LIN {X 0,Y 356.775,Z 285.085,A -85,B 0,C 180,E1 -13424.838,E2 -13424.838} C_VEL
LIN {X 0,Y 357.829,Z 274.843,A -85,B 0,C 180,E1 -13426.253,E2 -13426.253} C_VEL
LIN {X 0,Y 359.129,Z 263.368,A -85,B 0,C 180,E1 -13427.511,E2 -13427.511} C_VEL
LIN {X 0,Y 359.899,Z 254.34,A -85,B 0,C 180,E1 -13428.318,E2 -13428.318} C_VEL
LIN {X 0,Y 358.765,Z 242.212,A -85,B 0,C 180,E1 -13429.298,E2 -13429.298} C_VEL
LIN {X 0,Y 357.108,Z 229.36,A -85,B 0,C 180,E1 -13430.125,E2 -13430.125} C_VEL
LIN {X 0,Y 354.791,Z 217.977,A -85,B 0,C 180,E1 -13430.723,E2 -13430.723} C_VEL
LIN {X 0,Y 354.42,Z 215.798,A -85,B 0,C 180,E1 -13430.814,E2 -13430.814} C_VEL
LIN {X 0,Y 355.129,Z 206.721,A -85,B 0,C 180,E1 -13435.182,E2 -13435.182} C_VEL
LIN {X 0,Y 355.876,Z 199.228,A -85,B 0,C 180,E1 -13438.937,E2 -13438.937} C_VEL
LIN {X 0,Y 356.784,Z 191.893,A -85,B 0,C 180,E1 -13442.8,E2 -13442.8} C_VEL
LIN {X 0,Y 357.544,Z 185.922,A -85,B 0,C 180,E1 -13446.135,E2 -13446.135} C_VEL
LIN {X 0,Y 357.42,Z 182.644,A -85,B 0,C 180,E1 -13448.137,E2 -13448.137} C_VEL
LIN {X 0,Y 356.521,Z 177.676,A -85,B 0,C 180,E1 -13451.488,E2 -13451.488} C_VEL
LIN {X 0,Y 355.708,Z 173.412,A -85,B 0,C 180,E1 -13454.66,E2 -13454.66} C_VEL
LIN {X 0,Y 355.078,Z 169.762,A -85,B 0,C 180,E1 -13457.704,E2 -13457.704} C_VEL
LIN {X 0,Y 354.793,Z 168.296,A -85,B 0,C 180,E1 -13459.179,E2 -13459.179} C_VEL
LIN {X 0,Y 354.812,Z 168.29,A -85,B 0,C 180,E1 -13462.402,E2 -13462.402} C_VEL
LIN {X 0,Y 354.816,Z 168.291,A -85,B 0,C 180,E1 -13464.941,E2 -13464.941} C_VEL
LIN {X 0,Y 354.797,Z 168.292,A -85,B 0,C 180,E1 -13468.405,E2 -13468.405} C_VEL
LIN {X 0,Y 354.852,Z 168.283,A -85,B 0,C 180,E1 -13471.619,E2 -13471.619} C_VEL
LIN {X 0,Y 354.904,Z 168.279,A -85,B 0,C 180,E1 -13474.172,E2 -13474.172} C_VEL
LIN {X 0,Y 354.839,Z 168.284,A -85,B 0,C 180,E1 -13477.894,E2 -13477.894} C_VEL
LIN {X 0,Y 354.894,Z 168.275,A -85,B 0,C 180,E1 -13481.907,E2 -13481.907} C_VEL
LIN {X 0,Y 354.947,Z 168.272,A -85,B 0,C 180,E1 -13485.981,E2 -13485.981} C_VEL
LIN {X 0,Y 354.982,Z 168.269,A -85,B 0,C 180,E1 -13489.735,E2 -13489.735} C_VEL
LIN {X 0,Y 355.119,Z 168.251,A -85,B 0,C 180,E1 -13492.036,E2 -13492.036} C_VEL
LIN {X 0,Y 355.097,Z 168.254,A -85,B 0,C 180,E1 -13494.32,E2 -13494.32} C_VEL
LIN {X 0,Y 355.25,Z 168.233,A -85,B 0,C 180,E1 -13497.732,E2 -13497.732} C_VEL
LIN {X 0,Y 355.402,Z 168.217,A -85,B 0,C 180,E1 -13499.999,E2 -13499.999} C_VEL
LIN {X 0,Y 355.249,Z 168.235,A -85,B 0,C 180,E1 -13502.267,E2 -13502.267} C_VEL
LIN {X 0,Y 355.12,Z 168.255,A -85,B 0,C 180,E1 -13506.819,E2 -13506.819} C_VEL
LIN {X 0,Y 355.051,Z 168.263,A -85,B 0,C 180,E1 -13508.221,E2 -13508.221} C_VEL
LIN {X 0,Y 354.9,Z 170.431,A -85,B 0,C 180,E1 -13511.421,E2 -13511.421} C_VEL
LIN {X 0,Y 354.8,Z 172.389,A -85,B 0,C 180,E1 -13513.924,E2 -13513.924} C_VEL
LIN {X 0,Y 354.539,Z 175.648,A -85,B 0,C 180,E1 -13517.917,E2 -13517.917} C_VEL
LIN {X 0,Y 354.304,Z 178.431,A -85,B 0,C 180,E1 -13521.203,E2 -13521.203} C_VEL
LIN {X 0,Y 354.202,Z 181.144,A -85,B 0,C 180,E1 -13524.252,E2 -13524.252} C_VEL
LIN {X 0,Y 358.527,Z 194.659,A -85,B 0,C 180,E1 -13525.158,E2 -13525.158} C_VEL
LIN {X 0,Y 361.477,Z 206.388,A -85,B 0,C 180,E1 -13526.096,E2 -13526.096} C_VEL
LIN {X 0,Y 361.751,Z 209.952,A -85,B 0,C 180,E1 -13526.385,E2 -13526.385} C_VEL
LIN {X 0,Y 360.756,Z 221.591,A -85,B 0,C 180,E1 -13527.355,E2 -13527.355} C_VEL
LIN {X 0,Y 359.616,Z 232.741,A -85,B 0,C 180,E1 -13528.548,E2 -13528.548} C_VEL
LIN {X 0,Y 358.455,Z 243.363,A -85,B 0,C 180,E1 -13529.979,E2 -13529.979} C_VEL
LIN {X 0,Y 357.405,Z 251.936,A -85,B 0,C 180,E1 -13531.405,E2 -13531.405} C_VEL
LIN {X 0,Y 356.49,Z 258.964,A -85,B 0,C 180,E1 -13532.828,E2 -13532.828} C_VEL
LIN {X 0,Y 355.584,Z 265.414,A -85,B 0,C 180,E1 -13534.421,E2 -13534.421} C_VEL
LIN {X 0,Y 354.814,Z 271.831,A -85,B 0,C 180,E1 -13536.457,E2 -13536.457} C_VEL
LIN {X 0,Y 354.316,Z 275.481,A -85,B 0,C 180,E1 -13537.944,E2 -13537.944} C_VEL
LIN {X 0,Y 353.932,Z 278.366,A -85,B 0,C 180,E1 -13539.45,E2 -13539.45} C_VEL
LIN {X 0,Y 353.666,Z 280.464,A -85,B 0,C 180,E1 -13540.977,E2 -13540.977} C_VEL
LIN {X 0,Y 353.412,Z 281.894,A -85,B 0,C 180,E1 -13542.626,E2 -13542.626} C_VEL
LIN {X 0,Y 353.307,Z 282.48,A -85,B 0,C 180,E1 -13544.265,E2 -13544.265} C_VEL
LIN {X 0,Y 353.269,Z 282.265,A -85,B 0,C 180,E1 -13545.869,E2 -13545.869} C_VEL
LIN {X 0,Y 353.343,Z 281.274,A -85,B 0,C 180,E1 -13547.447,E2 -13547.447} C_VEL
LIN {X 0,Y 353.601,Z 279.433,A -85,B 0,C 180,E1 -13549.048,E2 -13549.048} C_VEL
LIN {X 0,Y 353.884,Z 276.549,A -85,B 0,C 180,E1 -13550.761,E2 -13550.761} C_VEL
LIN {X 0,Y 354.254,Z 272.517,A -85,B 0,C 180,E1 -13552.518,E2 -13552.518} C_VEL
LIN {X 0,Y 354.804,Z 267.177,A -85,B 0,C 180,E1 -13554.304,E2 -13554.304} C_VEL
LIN {X 0,Y 355.491,Z 260.179,A -85,B 0,C 180,E1 -13556.132,E2 -13556.132} C_VEL
LIN {X 0,Y 356.46,Z 251.262,A -85,B 0,C 180,E1 -13557.971,E2 -13557.971} C_VEL
LIN {X 0,Y 357.381,Z 242.57,A -85,B 0,C 180,E1 -13559.412,E2 -13559.412} C_VEL
LIN {X 0,Y 358.284,Z 232.446,A -85,B 0,C 180,E1 -13560.775,E2 -13560.775} C_VEL
LIN {X 0,Y 359.268,Z 221.132,A -85,B 0,C 180,E1 -13561.999,E2 -13561.999} C_VEL
LIN {X 0,Y 360.173,Z 210.079,A -85,B 0,C 180,E1 -13562.942,E2 -13562.942} C_VEL
LIN {X 0,Y 360.394,Z 206.56,A -85,B 0,C 180,E1 -13563.195,E2 -13563.195} C_VEL
LIN {X 0,Y 357.934,Z 194.376,A -85,B 0,C 180,E1 -13564.095,E2 -13564.095} C_VEL
LIN {X 0,Y 354.563,Z 181.298,A -85,B 0,C 180,E1 -13564.854,E2 -13564.854} C_VEL
LIN {X 0,Y 353.903,Z 178.558,A -85,B 0,C 180,E1 -13565,E2 -13565} C_VEL
LIN {X 0,Y 353.948,Z 174.587,A -85,B 0,C 180,E1 -13569.059,E2 -13569.059} C_VEL
LIN {X 0,Y 354.121,Z 171.115,A -85,B 0,C 180,E1 -13572.681,E2 -13572.681} C_VEL
LIN {X 0,Y 354.212,Z 168.881,A -85,B 0,C 180,E1 -13575.052,E2 -13575.052} C_VEL
LIN {X 0,Y 354.375,Z 168.346,A -85,B 0,C 180,E1 -13576.351,E2 -13576.351} C_VEL
LIN {X 0,Y 354.77,Z 168.292,A -85,B 0,C 180,E1 -13579.73,E2 -13579.73} C_VEL
LIN {X 0,Y 355.057,Z 168.26,A -85,B 0,C 180,E1 -13582.035,E2 -13582.035} C_VEL
LIN {X 0,Y 355.08,Z 168.257,A -85,B 0,C 180,E1 -13584.32,E2 -13584.32} C_VEL
LIN {X 0,Y 355.243,Z 168.235,A -85,B 0,C 180,E1 -13587.732,E2 -13587.732} C_VEL
LIN {X 0,Y 355.395,Z 168.218,A -85,B 0,C 180,E1 -13590,E2 -13590} C_VEL
LIN {X 0,Y 355.243,Z 168.235,A -85,B 0,C 180,E1 -13592.267,E2 -13592.267} C_VEL
LIN {X 0,Y 355.134,Z 168.246,A -85,B 0,C 180,E1 -13596.819,E2 -13596.819} C_VEL
LIN {X 0,Y 355.012,Z 168.261,A -85,B 0,C 180,E1 -13599.112,E2 -13599.112} C_VEL
LIN {X 0,Y 354.918,Z 168.272,A -85,B 0,C 180,E1 -13602.581,E2 -13602.581} C_VEL
LIN {X 0,Y 354.886,Z 168.279,A -85,B 0,C 180,E1 -13606.096,E2 -13606.096} C_VEL
LIN {X 0,Y 354.898,Z 168.275,A -85,B 0,C 180,E1 -13608.472,E2 -13608.472} C_VEL
LIN {X 0,Y 354.831,Z 168.284,A -85,B 0,C 180,E1 -13612.106,E2 -13612.106} C_VEL
LIN {X 0,Y 354.896,Z 168.278,A -85,B 0,C 180,E1 -13615.828,E2 -13615.828} C_VEL
LIN {X 0,Y 354.814,Z 168.288,A -85,B 0,C 180,E1 -13619.682,E2 -13619.682} C_VEL
LIN {X 0,Y 354.803,Z 168.289,A -85,B 0,C 180,E1 -13623.702,E2 -13623.702} C_VEL
LIN {X 0,Y 354.794,Z 168.288,A -85,B 0,C 180,E1 -13626.46,E2 -13626.46} C_VEL
LIN {X 0,Y 354.821,Z 168.288,A -85,B 0,C 180,E1 -13629.424,E2 -13629.424} C_VEL
LIN {X 0,Y 354.774,Z 168.291,A -85,B 0,C 180,E1 -13630.4,E2 -13630.4} C_VEL
LIN {X 0,Y 354.126,Z 168.376,A -85,B 0,C 180,E1 -13631.348,E2 -13631.348} C_VEL
LIN {X 0,Y 351.305,Z 168.731,A -85,B 0,C 180,E1 -13632.889,E2 -13632.889} C_VEL
LIN {X 0,Y 348.891,Z 169.031,A -85,B 0,C 180,E1 -13634.136,E2 -13634.136} C_VEL
LIN {X 0,Y 347.828,Z 169.161,A -85,B 0,C 180,E1 -13635.1,E2 -13635.1} C_VEL
LIN {X 0,Y 347.728,Z 169.169,A -85,B 0,C 180,E1 -13635.427,E2 -13635.427} C_VEL
LIN {X 0,Y 347.748,Z 169.167,A -85,B 0,C 180,E1 -13638.398,E2 -13638.398} C_VEL
LIN {X 0,Y 347.772,Z 169.162,A -85,B 0,C 180,E1 -13642.012,E2 -13642.012} C_VEL
LIN {X 0,Y 347.743,Z 169.166,A -85,B 0,C 180,E1 -13645.537,E2 -13645.537} C_VEL
LIN {X 0,Y 347.743,Z 169.168,A -85,B 0,C 180,E1 -13648.301,E2 -13648.301} C_VEL
LIN {X 0,Y 347.777,Z 169.165,A -85,B 0,C 180,E1 -13650.988,E2 -13650.988} C_VEL
LIN {X 0,Y 347.83,Z 169.155,A -85,B 0,C 180,E1 -13653.608,E2 -13653.608} C_VEL
LIN {X 0,Y 347.788,Z 169.162,A -85,B 0,C 180,E1 -13656.163,E2 -13656.163} C_VEL
LIN {X 0,Y 347.812,Z 169.158,A -85,B 0,C 180,E1 -13659.91,E2 -13659.91} C_VEL
LIN {X 0,Y 347.866,Z 169.156,A -85,B 0,C 180,E1 -13662.36,E2 -13662.36} C_VEL
LIN {X 0,Y 347.897,Z 169.149,A -85,B 0,C 180,E1 -13665.971,E2 -13665.971} C_VEL
LIN {X 0,Y 347.929,Z 169.143,A -85,B 0,C 180,E1 -13669.526,E2 -13669.526} C_VEL
LIN {X 0,Y 348.089,Z 169.123,A -85,B 0,C 180,E1 -13673.043,E2 -13673.043} C_VEL
LIN {X 0,Y 348.209,Z 169.11,A -85,B 0,C 180,E1 -13677.687,E2 -13677.687} C_VEL
LIN {X 0,Y 348.346,Z 169.096,A -85,B 0,C 180,E1 -13680.001,E2 -13680.001} C_VEL
LIN {X 0,Y 348.207,Z 169.111,A -85,B 0,C 180,E1 -13682.314,E2 -13682.314} C_VEL
LIN {X 0,Y 348.069,Z 169.125,A -85,B 0,C 180,E1 -13686.959,E2 -13686.959} C_VEL
LIN {X 0,Y 347.898,Z 169.147,A -85,B 0,C 180,E1 -13690.476,E2 -13690.476} C_VEL
LIN {X 0,Y 347.9,Z 169.149,A -85,B 0,C 180,E1 -13694.15,E2 -13694.15} C_VEL
LIN {X 0,Y 347.893,Z 169.148,A -85,B 0,C 180,E1 -13698.291,E2 -13698.291} C_VEL
LIN {X 0,Y 347.791,Z 169.165,A -85,B 0,C 180,E1 -13701.636,E2 -13701.636} C_VEL
LIN {X 0,Y 347.815,Z 169.159,A -85,B 0,C 180,E1 -13705.109,E2 -13705.109} C_VEL
LIN {X 0,Y 347.81,Z 169.161,A -85,B 0,C 180,E1 -13707.695,E2 -13707.695} C_VEL
LIN {X 0,Y 347.751,Z 169.165,A -85,B 0,C 180,E1 -13710.348,E2 -13710.348} C_VEL
LIN {X 0,Y 347.75,Z 169.166,A -85,B 0,C 180,E1 -13714.044,E2 -13714.044} C_VEL
LIN {X 0,Y 347.763,Z 169.169,A -85,B 0,C 180,E1 -13717.321,E2 -13717.321} C_VEL
LIN {X 0,Y 347.735,Z 169.17,A -85,B 0,C 180,E1 -13720.297,E2 -13720.297} C_VEL
LIN {X 0,Y 347.771,Z 169.229,A -85,B 0,C 180,E1 -13723.095,E2 -13723.095} C_VEL
LIN {X 0,Y 348.786,Z 174.756,A -85,B 0,C 180,E1 -13726.757,E2 -13726.757} C_VEL
LIN {X 0,Y 349.766,Z 179.946,A -85,B 0,C 180,E1 -13729.985,E2 -13729.985} C_VEL
LIN {X 0,Y 350.483,Z 185.084,A -85,B 0,C 180,E1 -13733.018,E2 -13733.018} C_VEL
LIN {X 0,Y 350.036,Z 190.177,A -85,B 0,C 180,E1 -13735.793,E2 -13735.793} C_VEL
LIN {X 0,Y 349.45,Z 195.261,A -85,B 0,C 180,E1 -13738.473,E2 -13738.473} C_VEL
LIN {X 0,Y 348.567,Z 203.172,A -85,B 0,C 180,E1 -13742.519,E2 -13742.519} C_VEL
LIN {X 0,Y 347.845,Z 210.499,A -85,B 0,C 180,E1 -13746.166,E2 -13746.166} C_VEL
LIN {X 0,Y 347.35,Z 216.92,A -85,B 0,C 180,E1 -13749.285,E2 -13749.285} C_VEL
LIN {X 0,Y 349.781,Z 231.182,A -85,B 0,C 180,E1 -13749.964,E2 -13749.964} C_VEL
LIN {X 0,Y 351.546,Z 244.711,A -85,B 0,C 180,E1 -13750.84,E2 -13750.84} C_VEL
LIN {X 0,Y 352.597,Z 257.024,A -85,B 0,C 180,E1 -13751.854,E2 -13751.854} C_VEL
LIN {X 0,Y 351.307,Z 268.693,A -85,B 0,C 180,E1 -13752.988,E2 -13752.988} C_VEL
LIN {X 0,Y 350.198,Z 279.222,A -85,B 0,C 180,E1 -13754.28,E2 -13754.28} C_VEL
LIN {X 0,Y 349.215,Z 288.757,A -85,B 0,C 180,E1 -13755.728,E2 -13755.728} C_VEL
LIN {X 0,Y 348.128,Z 297.936,A -85,B 0,C 180,E1 -13757.466,E2 -13757.466} C_VEL
LIN {X 0,Y 347.346,Z 305.337,A -85,B 0,C 180,E1 -13759.213,E2 -13759.213} C_VEL
LIN {X 0,Y 346.736,Z 312.139,A -85,B 0,C 180,E1 -13761.256,E2 -13761.256} C_VEL
LIN {X 0,Y 346.421,Z 316.621,A -85,B 0,C 180,E1 -13763.009,E2 -13763.009} C_VEL
LIN {X 0,Y 346.339,Z 318.984,A -85,B 0,C 180,E1 -13764.177,E2 -13764.177} C_VEL
LIN {X 0,Y 346.274,Z 320.909,A -85,B 0,C 180,E1 -13765.344,E2 -13765.344} C_VEL
LIN {X 0,Y 346.199,Z 322.391,A -85,B 0,C 180,E1 -13766.509,E2 -13766.509} C_VEL
LIN {X 0,Y 346.315,Z 324.064,A -85,B 0,C 180,E1 -13768.837,E2 -13768.837} C_VEL
LIN {X 0,Y 346.343,Z 324.305,A -85,B 0,C 180,E1 -13770,E2 -13770} C_VEL
LIN {X 0,Y 346.313,Z 324.129,A -85,B 0,C 180,E1 -13771.163,E2 -13771.163} C_VEL
LIN {X 0,Y 346.203,Z 322.506,A -85,B 0,C 180,E1 -13773.492,E2 -13773.492} C_VEL
LIN {X 0,Y 346.254,Z 321.099,A -85,B 0,C 180,E1 -13774.657,E2 -13774.657} C_VEL
LIN {X 0,Y 346.331,Z 318.743,A -85,B 0,C 180,E1 -13776.093,E2 -13776.093} C_VEL
LIN {X 0,Y 346.593,Z 314.163,A -85,B 0,C 180,E1 -13778.16,E2 -13778.16} C_VEL
LIN {X 0,Y 347.07,Z 309.057,A -85,B 0,C 180,E1 -13779.911,E2 -13779.911} C_VEL
LIN {X 0,Y 347.694,Z 302.672,A -85,B 0,C 180,E1 -13781.662,E2 -13781.662} C_VEL
LIN {X 0,Y 348.718,Z 294.729,A -85,B 0,C 180,E1 -13783.401,E2 -13783.401} C_VEL
LIN {X 0,Y 349.878,Z 284.878,A -85,B 0,C 180,E1 -13785.137,E2 -13785.137} C_VEL
LIN {X 0,Y 350.985,Z 274.712,A -85,B 0,C 180,E1 -13786.579,E2 -13786.579} C_VEL
LIN {X 0,Y 352.367,Z 263.307,A -85,B 0,C 180,E1 -13787.858,E2 -13787.858} C_VEL
LIN {X 0,Y 353.1,Z 255.693,A -85,B 0,C 180,E1 -13788.57,E2 -13788.57} C_VEL
LIN {X 0,Y 352.063,Z 243.656,A -85,B 0,C 180,E1 -13789.592,E2 -13789.592} C_VEL
LIN {X 0,Y 350.385,Z 229.904,A -85,B 0,C 180,E1 -13790.533,E2 -13790.533} C_VEL
LIN {X 0,Y 347.952,Z 217.951,A -85,B 0,C 180,E1 -13791.202,E2 -13791.202} C_VEL
LIN {X 0,Y 347.441,Z 215.266,A -85,B 0,C 180,E1 -13791.353,E2 -13791.353} C_VEL
LIN {X 0,Y 348.161,Z 206.443,A -85,B 0,C 180,E1 -13795.722,E2 -13795.722} C_VEL
LIN {X 0,Y 348.945,Z 199.183,A -85,B 0,C 180,E1 -13799.473,E2 -13799.473} C_VEL
LIN {X 0,Y 349.77,Z 192.92,A -85,B 0,C 180,E1 -13802.856,E2 -13802.856} C_VEL
LIN {X 0,Y 350.435,Z 188.155,A -85,B 0,C 180,E1 -13805.563,E2 -13805.563} C_VEL
LIN {X 0,Y 350.634,Z 185.806,A -85,B 0,C 180,E1 -13806.964,E2 -13806.964} C_VEL
LIN {X 0,Y 349.985,Z 181.224,A -85,B 0,C 180,E1 -13809.985,E2 -13809.985} C_VEL
LIN {X 0,Y 349.089,Z 176.365,A -85,B 0,C 180,E1 -13813.55,E2 -13813.55} C_VEL
LIN {X 0,Y 348.395,Z 172.498,A -85,B 0,C 180,E1 -13816.696,E2 -13816.696} C_VEL
LIN {X 0,Y 347.749,Z 169.173,A -85,B 0,C 180,E1 -13819.986,E2 -13819.986} C_VEL
LIN {X 0,Y 347.766,Z 169.168,A -85,B 0,C 180,E1 -13822.679,E2 -13822.679} C_VEL
LIN {X 0,Y 347.752,Z 169.167,A -85,B 0,C 180,E1 -13825.956,E2 -13825.956} C_VEL
LIN {X 0,Y 347.753,Z 169.167,A -85,B 0,C 180,E1 -13829.652,E2 -13829.652} C_VEL
LIN {X 0,Y 347.836,Z 169.157,A -85,B 0,C 180,E1 -13833.607,E2 -13833.607} C_VEL
LIN {X 0,Y 347.793,Z 169.164,A -85,B 0,C 180,E1 -13836.162,E2 -13836.162} C_VEL
LIN {X 0,Y 347.816,Z 169.158,A -85,B 0,C 180,E1 -13839.909,E2 -13839.909} C_VEL
LIN {X 0,Y 347.836,Z 169.158,A -85,B 0,C 180,E1 -13843.568,E2 -13843.568} C_VEL
LIN {X 0,Y 347.894,Z 169.151,A -85,B 0,C 180,E1 -13847.16,E2 -13847.16} C_VEL
LIN {X 0,Y 348.098,Z 169.126,A -85,B 0,C 180,E1 -13851.612,E2 -13851.612} C_VEL
LIN {X 0,Y 348.072,Z 169.129,A -85,B 0,C 180,E1 -13854.205,E2 -13854.205} C_VEL
LIN {X 0,Y 348.212,Z 169.11,A -85,B 0,C 180,E1 -13857.686,E2 -13857.686} C_VEL
LIN {X 0,Y 348.371,Z 169.093,A -85,B 0,C 180,E1 -13859.999,E2 -13859.999} C_VEL
LIN {X 0,Y 348.211,Z 169.111,A -85,B 0,C 180,E1 -13862.313,E2 -13862.313} C_VEL
LIN {X 0,Y 348.084,Z 169.132,A -85,B 0,C 180,E1 -13866.957,E2 -13866.957} C_VEL
LIN {X 0,Y 348.017,Z 169.275,A -85,B 0,C 180,E1 -13868.297,E2 -13868.297} C_VEL
LIN {X 0,Y 347.868,Z 171.74,A -85,B 0,C 180,E1 -13871.655,E2 -13871.655} C_VEL
LIN {X 0,Y 347.658,Z 174.513,A -85,B 0,C 180,E1 -13875.236,E2 -13875.236} C_VEL
LIN {X 0,Y 347.409,Z 177.461,A -85,B 0,C 180,E1 -13878.885,E2 -13878.885} C_VEL
LIN {X 0,Y 347.196,Z 180.611,A -85,B 0,C 180,E1 -13882.618,E2 -13882.618} C_VEL
LIN {X 0,Y 347.146,Z 181.545,A -85,B 0,C 180,E1 -13883.726,E2 -13883.726} C_VEL
LIN {X 0,Y 351.861,Z 196.051,A -85,B 0,C 180,E1 -13884.76,E2 -13884.76} C_VEL
LIN {X 0,Y 354.594,Z 206.767,A -85,B 0,C 180,E1 -13885.654,E2 -13885.654} C_VEL
LIN {X 0,Y 355.164,Z 210.24,A -85,B 0,C 180,E1 -13885.964,E2 -13885.964} C_VEL
LIN {X 0,Y 354.161,Z 221.531,A -85,B 0,C 180,E1 -13886.919,E2 -13886.919} C_VEL
LIN {X 0,Y 352.993,Z 232.201,A -85,B 0,C 180,E1 -13888.057,E2 -13888.057} C_VEL
LIN {X 0,Y 351.818,Z 242.651,A -85,B 0,C 180,E1 -13889.465,E2 -13889.465} C_VEL
LIN {X 0,Y 350.677,Z 251.567,A -85,B 0,C 180,E1 -13890.943,E2 -13890.943} C_VEL
LIN {X 0,Y 349.563,Z 259.723,A -85,B 0,C 180,E1 -13892.613,E2 -13892.613} C_VEL
LIN {X 0,Y 348.549,Z 266.572,A -85,B 0,C 180,E1 -13894.372,E2 -13894.372} C_VEL
LIN {X 0,Y 347.892,Z 271.876,A -85,B 0,C 180,E1 -13896.092,E2 -13896.092} C_VEL
LIN {X 0,Y 347.27,Z 276.182,A -85,B 0,C 180,E1 -13897.882,E2 -13897.882} C_VEL
LIN {X 0,Y 346.817,Z 279.319,A -85,B 0,C 180,E1 -13899.642,E2 -13899.642} C_VEL
LIN {X 0,Y 346.395,Z 282.009,A -85,B 0,C 180,E1 -13902.03,E2 -13902.03} C_VEL
LIN {X 0,Y 346.221,Z 282.824,A -85,B 0,C 180,E1 -13903.643,E2 -13903.643} C_VEL
LIN {X 0,Y 346.188,Z 282.856,A -85,B 0,C 180,E1 -13905.278,E2 -13905.278} C_VEL
LIN {X 0,Y 346.223,Z 282.083,A -85,B 0,C 180,E1 -13906.95,E2 -13906.95} C_VEL
LIN {X 0,Y 346.442,Z 280.448,A -85,B 0,C 180,E1 -13908.64,E2 -13908.64} C_VEL
LIN {X 0,Y 346.75,Z 277.852,A -85,B 0,C 180,E1 -13910.37,E2 -13910.37} C_VEL
LIN {X 0,Y 347.191,Z 272.99,A -85,B 0,C 180,E1 -13912.607,E2 -13912.607} C_VEL
LIN {X 0,Y 347.788,Z 267.492,A -85,B 0,C 180,E1 -13914.481,E2 -13914.481} C_VEL
LIN {X 0,Y 348.57,Z 260.05,A -85,B 0,C 180,E1 -13916.438,E2 -13916.438} C_VEL
LIN {X 0,Y 349.469,Z 252.131,A -85,B 0,C 180,E1 -13918.099,E2 -13918.099} C_VEL
LIN {X 0,Y 350.485,Z 242.782,A -85,B 0,C 180,E1 -13919.685,E2 -13919.685} C_VEL
LIN {X 0,Y 351.503,Z 231.908,A -85,B 0,C 180,E1 -13921.16,E2 -13921.16} C_VEL
LIN {X 0,Y 352.522,Z 220.586,A -85,B 0,C 180,E1 -13922.385,E2 -13922.385} C_VEL
LIN {X 0,Y 353.459,Z 209.14,A -85,B 0,C 180,E1 -13923.35,E2 -13923.35} C_VEL
LIN {X 0,Y 353.409,Z 206.39,A -85,B 0,C 180,E1 -13923.564,E2 -13923.564} C_VEL
LIN {X 0,Y 350.792,Z 194.106,A -85,B 0,C 180,E1 -13924.485,E2 -13924.485} C_VEL
LIN {X 0,Y 347.269,Z 180.844,A -85,B 0,C 180,E1 -13925.271,E2 -13925.271} C_VEL
LIN {X 0,Y 346.843,Z 178.951,A -85,B 0,C 180,E1 -13925.372,E2 -13925.372} C_VEL
LIN {X 0,Y 346.887,Z 175.681,A -85,B 0,C 180,E1 -13928.742,E2 -13928.742} C_VEL
LIN {X 0,Y 347.037,Z 172.294,A -85,B 0,C 180,E1 -13932.315,E2 -13932.315} C_VEL
LIN {X 0,Y 347.143,Z 170.03,A -85,B 0,C 180,E1 -13934.74,E2 -13934.74} C_VEL
LIN {X 0,Y 347.318,Z 169.225,A -85,B 0,C 180,E1 -13936.233,E2 -13936.233} C_VEL
LIN {X 0,Y 347.705,Z 169.171,A -85,B 0,C 180,E1 -13939.519,E2 -13939.519} C_VEL
LIN {X 0,Y 348.02,Z 169.134,A -85,B 0,C 180,E1 -13941.873,E2 -13941.873} C_VEL
LIN {X 0,Y 348.054,Z 169.132,A -85,B 0,C 180,E1 -13944.205,E2 -13944.205} C_VEL
LIN {X 0,Y 348.205,Z 169.111,A -85,B 0,C 180,E1 -13947.686,E2 -13947.686} C_VEL
LIN {X 0,Y 348.364,Z 169.094,A -85,B 0,C 180,E1 -13950,E2 -13950} C_VEL
LIN {X 0,Y 348.205,Z 169.111,A -85,B 0,C 180,E1 -13952.313,E2 -13952.313} C_VEL
LIN {X 0,Y 348.102,Z 169.121,A -85,B 0,C 180,E1 -13956.958,E2 -13956.958} C_VEL
LIN {X 0,Y 347.964,Z 169.14,A -85,B 0,C 180,E1 -13959.298,E2 -13959.298} C_VEL
LIN {X 0,Y 347.887,Z 169.148,A -85,B 0,C 180,E1 -13962.839,E2 -13962.839} C_VEL
LIN {X 0,Y 347.836,Z 169.155,A -85,B 0,C 180,E1 -13966.431,E2 -13966.431} C_VEL
LIN {X 0,Y 347.848,Z 169.153,A -85,B 0,C 180,E1 -13968.861,E2 -13968.861} C_VEL
LIN {X 0,Y 347.771,Z 169.162,A -85,B 0,C 180,E1 -13972.579,E2 -13972.579} C_VEL
LIN {X 0,Y 347.809,Z 169.16,A -85,B 0,C 180,E1 -13975.109,E2 -13975.109} C_VEL
LIN {X 0,Y 347.805,Z 169.161,A -85,B 0,C 180,E1 -13977.694,E2 -13977.694} C_VEL
LIN {X 0,Y 347.746,Z 169.166,A -85,B 0,C 180,E1 -13980.348,E2 -13980.348} C_VEL
LIN {X 0,Y 347.745,Z 169.166,A -85,B 0,C 180,E1 -13984.044,E2 -13984.044} C_VEL
LIN {X 0,Y 347.758,Z 169.169,A -85,B 0,C 180,E1 -13987.321,E2 -13987.321} C_VEL
LIN {X 0,Y 347.725,Z 169.168,A -85,B 0,C 180,E1 -13990.392,E2 -13990.392} C_VEL
LIN {X 0,Y 347.723,Z 169.171,A -85,B 0,C 180,E1 -13993.408,E2 -13993.408} C_VEL
LIN {X 0,Y 347.728,Z 169.169,A -85,B 0,C 180,E1 -13995.427,E2 -13995.427} C_VEL
LIN {X 0,Y 347.03,Z 169.257,A -85,B 0,C 180,E1 -13996.394,E2 -13996.394} C_VEL
LIN {X 0,Y 344.191,Z 169.608,A -85,B 0,C 180,E1 -13997.968,E2 -13997.968} C_VEL
LIN {X 0,Y 341.802,Z 169.909,A -85,B 0,C 180,E1 -13999.242,E2 -13999.242} C_VEL
LIN {X 0,Y 340.771,Z 170.035,A -85,B 0,C 180,E1 -14000.227,E2 -14000.227} C_VEL
LIN {X 0,Y 340.682,Z 170.044,A -85,B 0,C 180,E1 -14000.56,E2 -14000.56} C_VEL
LIN {X 0,Y 340.708,Z 170.042,A -85,B 0,C 180,E1 -14003.56,E2 -14003.56} C_VEL
LIN {X 0,Y 340.69,Z 170.045,A -85,B 0,C 180,E1 -14006.154,E2 -14006.154} C_VEL
LIN {X 0,Y 340.74,Z 170.04,A -85,B 0,C 180,E1 -14010.33,E2 -14010.33} C_VEL
LIN {X 0,Y 340.802,Z 170.033,A -85,B 0,C 180,E1 -14013.021,E2 -14013.021} C_VEL
LIN {X 0,Y 340.729,Z 170.042,A -85,B 0,C 180,E1 -14016.928,E2 -14016.928} C_VEL
LIN {X 0,Y 340.79,Z 170.035,A -85,B 0,C 180,E1 -14020.734,E2 -14020.734} C_VEL
LIN {X 0,Y 340.786,Z 170.033,A -85,B 0,C 180,E1 -14023.219,E2 -14023.219} C_VEL
LIN {X 0,Y 340.844,Z 170.026,A -85,B 0,C 180,E1 -14026.891,E2 -14026.891} C_VEL
LIN {X 0,Y 340.914,Z 170.02,A -85,B 0,C 180,E1 -14030.508,E2 -14030.508} C_VEL
LIN {X 0,Y 341.057,Z 169.999,A -85,B 0,C 180,E1 -14032.898,E2 -14032.898} C_VEL
LIN {X 0,Y 341.171,Z 169.986,A -85,B 0,C 180,E1 -14037.639,E2 -14037.639} C_VEL
LIN {X 0,Y 341.296,Z 169.974,A -85,B 0,C 180,E1 -14040.001,E2 -14040.001} C_VEL
LIN {X 0,Y 341.169,Z 169.987,A -85,B 0,C 180,E1 -14042.362,E2 -14042.362} C_VEL
LIN {X 0,Y 341.017,Z 170.004,A -85,B 0,C 180,E1 -14047.104,E2 -14047.104} C_VEL
LIN {X 0,Y 340.85,Z 170.024,A -85,B 0,C 180,E1 -14050.695,E2 -14050.695} C_VEL
LIN {X 0,Y 340.865,Z 170.024,A -85,B 0,C 180,E1 -14054.325,E2 -14054.325} C_VEL
LIN {X 0,Y 340.84,Z 170.026,A -85,B 0,C 180,E1 -14058.467,E2 -14058.467} C_VEL
LIN {X 0,Y 340.756,Z 170.039,A -85,B 0,C 180,E1 -14061.857,E2 -14061.857} C_VEL
LIN {X 0,Y 340.775,Z 170.038,A -85,B 0,C 180,E1 -14065.665,E2 -14065.665} C_VEL
LIN {X 0,Y 340.73,Z 170.039,A -85,B 0,C 180,E1 -14068.321,E2 -14068.321} C_VEL
LIN {X 0,Y 340.7,Z 170.046,A -85,B 0,C 180,E1 -14071.045,E2 -14071.045} C_VEL
LIN {X 0,Y 340.72,Z 170.046,A -85,B 0,C 180,E1 -14075.279,E2 -14075.279} C_VEL
LIN {X 0,Y 340.711,Z 170.045,A -85,B 0,C 180,E1 -14078.386,E2 -14078.386} C_VEL
LIN {X 0,Y 340.727,Z 170.039,A -85,B 0,C 180,E1 -14082.42,E2 -14082.42} C_VEL
LIN {X 0,Y 340.769,Z 170.357,A -85,B 0,C 180,E1 -14082.891,E2 -14082.891} C_VEL
LIN {X 0,Y 341.632,Z 175.023,A -85,B 0,C 180,E1 -14086.056,E2 -14086.056} C_VEL
LIN {X 0,Y 342.595,Z 180.193,A -85,B 0,C 180,E1 -14089.379,E2 -14089.379} C_VEL
LIN {X 0,Y 343.314,Z 184.683,A -85,B 0,C 180,E1 -14092.111,E2 -14092.111} C_VEL
LIN {X 0,Y 343.34,Z 188.52,A -85,B 0,C 180,E1 -14094.312,E2 -14094.312} C_VEL
LIN {X 0,Y 342.567,Z 194.872,A -85,B 0,C 180,E1 -14097.764,E2 -14097.764} C_VEL
LIN {X 0,Y 341.664,Z 202.479,A -85,B 0,C 180,E1 -14101.764,E2 -14101.764} C_VEL
LIN {X 0,Y 340.868,Z 210.052,A -85,B 0,C 180,E1 -14105.647,E2 -14105.647} C_VEL
LIN {X 0,Y 340.355,Z 216.787,A -85,B 0,C 180,E1 -14108.907,E2 -14108.907} C_VEL
LIN {X 0,Y 342.72,Z 230.635,A -85,B 0,C 180,E1 -14109.576,E2 -14109.576} C_VEL
LIN {X 0,Y 344.481,Z 243.574,A -85,B 0,C 180,E1 -14110.431,E2 -14110.431} C_VEL
LIN {X 0,Y 345.675,Z 256.095,A -85,B 0,C 180,E1 -14111.478,E2 -14111.478} C_VEL
LIN {X 0,Y 344.595,Z 266.611,A -85,B 0,C 180,E1 -14112.493,E2 -14112.493} C_VEL
LIN {X 0,Y 343.407,Z 277.439,A -85,B 0,C 180,E1 -14113.809,E2 -14113.809} C_VEL
LIN {X 0,Y 342.514,Z 286.314,A -85,B 0,C 180,E1 -14115.139,E2 -14115.139} C_VEL
LIN {X 0,Y 341.558,Z 294.479,A -85,B 0,C 180,E1 -14116.616,E2 -14116.616} C_VEL
LIN {X 0,Y 340.549,Z 302.493,A -85,B 0,C 180,E1 -14118.392,E2 -14118.392} C_VEL
LIN {X 0,Y 340.059,Z 307.932,A -85,B 0,C 180,E1 -14119.883,E2 -14119.883} C_VEL
LIN {X 0,Y 339.548,Z 313.248,A -85,B 0,C 180,E1 -14121.669,E2 -14121.669} C_VEL
LIN {X 0,Y 339.298,Z 317.381,A -85,B 0,C 180,E1 -14123.459,E2 -14123.459} C_VEL
LIN {X 0,Y 339.193,Z 320.437,A -85,B 0,C 180,E1 -14125.246,E2 -14125.246} C_VEL
LIN {X 0,Y 339.124,Z 321.937,A -85,B 0,C 180,E1 -14126.436,E2 -14126.436} C_VEL
LIN {X 0,Y 339.222,Z 323.628,A -85,B 0,C 180,E1 -14128.813,E2 -14128.813} C_VEL
LIN {X 0,Y 339.284,Z 323.879,A -85,B 0,C 180,E1 -14130,E2 -14130} C_VEL
LIN {X 0,Y 339.219,Z 323.716,A -85,B 0,C 180,E1 -14131.187,E2 -14131.187} C_VEL
LIN {X 0,Y 339.126,Z 322.114,A -85,B 0,C 180,E1 -14133.565,E2 -14133.565} C_VEL
LIN {X 0,Y 339.174,Z 320.717,A -85,B 0,C 180,E1 -14134.755,E2 -14134.755} C_VEL
LIN {X 0,Y 339.279,Z 317.788,A -85,B 0,C 180,E1 -14136.542,E2 -14136.542} C_VEL
LIN {X 0,Y 339.549,Z 313.826,A -85,B 0,C 180,E1 -14138.331,E2 -14138.331} C_VEL
LIN {X 0,Y 340.058,Z 308.741,A -85,B 0,C 180,E1 -14140.118,E2 -14140.118} C_VEL
LIN {X 0,Y 340.703,Z 302.382,A -85,B 0,C 180,E1 -14141.905,E2 -14141.905} C_VEL
LIN {X 0,Y 341.788,Z 294.485,A -85,B 0,C 180,E1 -14143.678,E2 -14143.678} C_VEL
LIN {X 0,Y 342.787,Z 286.465,A -85,B 0,C 180,E1 -14145.154,E2 -14145.154} C_VEL
LIN {X 0,Y 344.02,Z 275.667,A -85,B 0,C 180,E1 -14146.772,E2 -14146.772} C_VEL
LIN {X 0,Y 345.439,Z 264.686,A -85,B 0,C 180,E1 -14148.075,E2 -14148.075} C_VEL
LIN {X 0,Y 346.298,Z 257.332,A -85,B 0,C 180,E1 -14148.795,E2 -14148.795} C_VEL
LIN {X 0,Y 345.417,Z 245.496,A -85,B 0,C 180,E1 -14149.878,E2 -14149.878} C_VEL
LIN {X 0,Y 343.941,Z 232.35,A -85,B 0,C 180,E1 -14150.839,E2 -14150.839} C_VEL
LIN {X 0,Y 341.543,Z 219.961,A -85,B 0,C 180,E1 -14151.59,E2 -14151.59} C_VEL
LIN {X 0,Y 340.442,Z 214.776,A -85,B 0,C 180,E1 -14151.893,E2 -14151.893} C_VEL
LIN {X 0,Y 341.099,Z 207.419,A -85,B 0,C 180,E1 -14155.638,E2 -14155.638} C_VEL
LIN {X 0,Y 341.914,Z 200.013,A -85,B 0,C 180,E1 -14159.559,E2 -14159.559} C_VEL
LIN {X 0,Y 342.708,Z 194.212,A -85,B 0,C 180,E1 -14162.775,E2 -14162.775} C_VEL
LIN {X 0,Y 343.44,Z 189.192,A -85,B 0,C 180,E1 -14165.676,E2 -14165.676} C_VEL
LIN {X 0,Y 343.634,Z 186.923,A -85,B 0,C 180,E1 -14167.095,E2 -14167.095} C_VEL
LIN {X 0,Y 343.185,Z 183.447,A -85,B 0,C 180,E1 -14169.409,E2 -14169.409} C_VEL
LIN {X 0,Y 342.359,Z 179.033,A -85,B 0,C 180,E1 -14172.643,E2 -14172.643} C_VEL
LIN {X 0,Y 341.567,Z 174.817,A -85,B 0,C 180,E1 -14176.067,E2 -14176.067} C_VEL
LIN {X 0,Y 340.879,Z 170.904,A -85,B 0,C 180,E1 -14179.716,E2 -14179.716} C_VEL
LIN {X 0,Y 340.702,Z 170.05,A -85,B 0,C 180,E1 -14180.616,E2 -14180.616} C_VEL
LIN {X 0,Y 340.714,Z 170.046,A -85,B 0,C 180,E1 -14183.559,E2 -14183.559} C_VEL
LIN {X 0,Y 340.696,Z 170.047,A -85,B 0,C 180,E1 -14186.153,E2 -14186.153} C_VEL
LIN {X 0,Y 340.745,Z 170.043,A -85,B 0,C 180,E1 -14190.329,E2 -14190.329} C_VEL
LIN {X 0,Y 340.808,Z 170.031,A -85,B 0,C 180,E1 -14193.02,E2 -14193.02} C_VEL
LIN {X 0,Y 340.733,Z 170.042,A -85,B 0,C 180,E1 -14196.927,E2 -14196.927} C_VEL
LIN {X 0,Y 340.769,Z 170.04,A -85,B 0,C 180,E1 -14200.732,E2 -14200.732} C_VEL
LIN {X 0,Y 340.821,Z 170.033,A -85,B 0,C 180,E1 -14204.45,E2 -14204.45} C_VEL
LIN {X 0,Y 340.854,Z 170.029,A -85,B 0,C 180,E1 -14208.1,E2 -14208.1} C_VEL
LIN {X 0,Y 341.045,Z 170.005,A -85,B 0,C 180,E1 -14211.706,E2 -14211.706} C_VEL
LIN {X 0,Y 341.048,Z 170.004,A -85,B 0,C 180,E1 -14214.085,E2 -14214.085} C_VEL
LIN {X 0,Y 341.174,Z 169.986,A -85,B 0,C 180,E1 -14217.638,E2 -14217.638} C_VEL
LIN {X 0,Y 341.32,Z 169.971,A -85,B 0,C 180,E1 -14219.999,E2 -14219.999} C_VEL
LIN {X 0,Y 341.173,Z 169.988,A -85,B 0,C 180,E1 -14222.361,E2 -14222.361} C_VEL
LIN {X 0,Y 341.051,Z 170.008,A -85,B 0,C 180,E1 -14227.102,E2 -14227.102} C_VEL
LIN {X 0,Y 341.017,Z 170.554,A -85,B 0,C 180,E1 -14228.415,E2 -14228.415} C_VEL
LIN {X 0,Y 340.85,Z 173.073,A -85,B 0,C 180,E1 -14231.899,E2 -14231.899} C_VEL
LIN {X 0,Y 340.715,Z 174.897,A -85,B 0,C 180,E1 -14234.331,E2 -14234.331} C_VEL
LIN {X 0,Y 340.442,Z 177.989,A -85,B 0,C 180,E1 -14238.265,E2 -14238.265} C_VEL
LIN {X 0,Y 340.191,Z 180.904,A -85,B 0,C 180,E1 -14241.83,E2 -14241.83} C_VEL
LIN {X 0,Y 340.134,Z 182.047,A -85,B 0,C 180,E1 -14243.195,E2 -14243.195} C_VEL
LIN {X 0,Y 344.777,Z 195.961,A -85,B 0,C 180,E1 -14244.228,E2 -14244.228} C_VEL
LIN {X 0,Y 348.032,Z 208.62,A -85,B 0,C 180,E1 -14245.325,E2 -14245.325} C_VEL
LIN {X 0,Y 348.477,Z 210.994,A -85,B 0,C 180,E1 -14245.552,E2 -14245.552} C_VEL
LIN {X 0,Y 347.492,Z 222.444,A -85,B 0,C 180,E1 -14246.551,E2 -14246.551} C_VEL
LIN {X 0,Y 346.284,Z 232.952,A -85,B 0,C 180,E1 -14247.704,E2 -14247.704} C_VEL
LIN {X 0,Y 345.149,Z 242.678,A -85,B 0,C 180,E1 -14249.038,E2 -14249.038} C_VEL
LIN {X 0,Y 344.04,Z 250.713,A -85,B 0,C 180,E1 -14250.37,E2 -14250.37} C_VEL
LIN {X 0,Y 343.037,Z 258.04,A -85,B 0,C 180,E1 -14251.839,E2 -14251.839} C_VEL
LIN {X 0,Y 341.813,Z 265.68,A -85,B 0,C 180,E1 -14253.72,E2 -14253.72} C_VEL
LIN {X 0,Y 341.167,Z 270.537,A -85,B 0,C 180,E1 -14255.225,E2 -14255.225} C_VEL
LIN {X 0,Y 340.585,Z 274.577,A -85,B 0,C 180,E1 -14256.756,E2 -14256.756} C_VEL
LIN {X 0,Y 340.081,Z 277.852,A -85,B 0,C 180,E1 -14258.313,E2 -14258.313} C_VEL
LIN {X 0,Y 339.661,Z 280.553,A -85,B 0,C 180,E1 -14260.041,E2 -14260.041} C_VEL
LIN {X 0,Y 339.347,Z 282.353,A -85,B 0,C 180,E1 -14261.791,E2 -14261.791} C_VEL
LIN {X 0,Y 339.145,Z 283.241,A -85,B 0,C 180,E1 -14263.506,E2 -14263.506} C_VEL
LIN {X 0,Y 339.101,Z 283.299,A -85,B 0,C 180,E1 -14265.197,E2 -14265.197} C_VEL
LIN {X 0,Y 339.128,Z 282.583,A -85,B 0,C 180,E1 -14266.852,E2 -14266.852} C_VEL
LIN {X 0,Y 339.339,Z 281.106,A -85,B 0,C 180,E1 -14268.49,E2 -14268.49} C_VEL
LIN {X 0,Y 339.621,Z 278.849,A -85,B 0,C 180,E1 -14270.096,E2 -14270.096} C_VEL
LIN {X 0,Y 339.933,Z 275.625,A -85,B 0,C 180,E1 -14271.778,E2 -14271.778} C_VEL
LIN {X 0,Y 340.432,Z 270.986,A -85,B 0,C 180,E1 -14273.622,E2 -14273.622} C_VEL
LIN {X 0,Y 341.061,Z 264.879,A -85,B 0,C 180,E1 -14275.511,E2 -14275.511} C_VEL
LIN {X 0,Y 341.987,Z 257.01,A -85,B 0,C 180,E1 -14277.411,E2 -14277.411} C_VEL
LIN {X 0,Y 343.097,Z 247.75,A -85,B 0,C 180,E1 -14279.196,E2 -14279.196} C_VEL
LIN {X 0,Y 344.093,Z 238.368,A -85,B 0,C 180,E1 -14280.646,E2 -14280.646} C_VEL
LIN {X 0,Y 345.055,Z 228.151,A -85,B 0,C 180,E1 -14281.933,E2 -14281.933} C_VEL
LIN {X 0,Y 346.017,Z 217.189,A -85,B 0,C 180,E1 -14283.045,E2 -14283.045} C_VEL
LIN {X 0,Y 346.662,Z 209.563,A -85,B 0,C 180,E1 -14283.674,E2 -14283.674} C_VEL
LIN {X 0,Y 345.953,Z 204.441,A -85,B 0,C 180,E1 -14284.099,E2 -14284.099} C_VEL
LIN {X 0,Y 343.026,Z 191.572,A -85,B 0,C 180,E1 -14285.043,E2 -14285.043} C_VEL
LIN {X 0,Y 339.766,Z 179.333,A -85,B 0,C 180,E1 -14285.766,E2 -14285.766} C_VEL
LIN {X 0,Y 339.835,Z 175.848,A -85,B 0,C 180,E1 -14289.416,E2 -14289.416} C_VEL
LIN {X 0,Y 340,Z 172.338,A -85,B 0,C 180,E1 -14293.178,E2 -14293.178} C_VEL
LIN {X 0,Y 340.171,Z 170.114,A -85,B 0,C 180,E1 -14295.645,E2 -14295.645} C_VEL
LIN {X 0,Y 340.633,Z 170.051,A -85,B 0,C 180,E1 -14299.298,E2 -14299.298} C_VEL
LIN {X 0,Y 340.952,Z 170.013,A -85,B 0,C 180,E1 -14301.704,E2 -14301.704} C_VEL
LIN {X 0,Y 341.029,Z 170.007,A -85,B 0,C 180,E1 -14304.085,E2 -14304.085} C_VEL
LIN {X 0,Y 341.167,Z 169.987,A -85,B 0,C 180,E1 -14307.639,E2 -14307.639} C_VEL
LIN {X 0,Y 341.313,Z 169.972,A -85,B 0,C 180,E1 -14310,E2 -14310} C_VEL
LIN {X 0,Y 341.167,Z 169.987,A -85,B 0,C 180,E1 -14312.361,E2 -14312.361} C_VEL
LIN {X 0,Y 341.071,Z 169.997,A -85,B 0,C 180,E1 -14317.102,E2 -14317.102} C_VEL
LIN {X 0,Y 340.868,Z 170.022,A -85,B 0,C 180,E1 -14320.694,E2 -14320.694} C_VEL
LIN {X 0,Y 340.859,Z 170.024,A -85,B 0,C 180,E1 -14324.325,E2 -14324.325} C_VEL
LIN {X 0,Y 340.833,Z 170.027,A -85,B 0,C 180,E1 -14328.466,E2 -14328.466} C_VEL
LIN {X 0,Y 340.75,Z 170.04,A -85,B 0,C 180,E1 -14331.857,E2 -14331.857} C_VEL
LIN {X 0,Y 340.769,Z 170.038,A -85,B 0,C 180,E1 -14335.665,E2 -14335.665} C_VEL
LIN {X 0,Y 340.725,Z 170.04,A -85,B 0,C 180,E1 -14338.321,E2 -14338.321} C_VEL
LIN {X 0,Y 340.694,Z 170.047,A -85,B 0,C 180,E1 -14341.045,E2 -14341.045} C_VEL
LIN {X 0,Y 340.715,Z 170.047,A -85,B 0,C 180,E1 -14345.279,E2 -14345.279} C_VEL
LIN {X 0,Y 340.707,Z 170.042,A -85,B 0,C 180,E1 -14348.386,E2 -14348.386} C_VEL
LIN {X 0,Y 340.696,Z 170.044,A -85,B 0,C 180,E1 -14352.046,E2 -14352.046} C_VEL
LIN {X 0,Y 340.68,Z 170.048,A -85,B 0,C 180,E1 -14355.462,E2 -14355.462} C_VEL
LIN {X 0,Y 340.684,Z 170.048,A -85,B 0,C 180,E1 -14358.691,E2 -14358.691} C_VEL
LIN {X 0,Y 340.682,Z 170.044,A -85,B 0,C 180,E1 -14360.56,E2 -14360.56} C_VEL
LIN {X 0,Y 340.01,Z 170.13,A -85,B 0,C 180,E1 -14361.548,E2 -14361.548} C_VEL
LIN {X 0,Y 337.184,Z 170.484,A -85,B 0,C 180,E1 -14363.155,E2 -14363.155} C_VEL
LIN {X 0,Y 334.783,Z 170.782,A -85,B 0,C 180,E1 -14364.456,E2 -14364.456} C_VEL
LIN {X 0,Y 333.733,Z 170.912,A -85,B 0,C 180,E1 -14365.462,E2 -14365.462} C_VEL
LIN {X 0,Y 333.637,Z 170.923,A -85,B 0,C 180,E1 -14365.803,E2 -14365.803} C_VEL
LIN {X 0,Y 333.693,Z 170.916,A -85,B 0,C 180,E1 -14369.713,E2 -14369.713} C_VEL
LIN {X 0,Y 333.738,Z 170.913,A -85,B 0,C 180,E1 -14372.401,E2 -14372.401} C_VEL
LIN {X 0,Y 333.726,Z 170.913,A -85,B 0,C 180,E1 -14375.091,E2 -14375.091} C_VEL
LIN {X 0,Y 333.684,Z 170.918,A -85,B 0,C 180,E1 -14379.02,E2 -14379.02} C_VEL
LIN {X 0,Y 333.793,Z 170.903,A -85,B 0,C 180,E1 -14381.59,E2 -14381.59} C_VEL
LIN {X 0,Y 333.808,Z 170.902,A -85,B 0,C 180,E1 -14385.577,E2 -14385.577} C_VEL
LIN {X 0,Y 333.834,Z 170.898,A -85,B 0,C 180,E1 -14389.079,E2 -14389.079} C_VEL
LIN {X 0,Y 334.005,Z 170.878,A -85,B 0,C 180,E1 -14392.748,E2 -14392.748} C_VEL
LIN {X 0,Y 333.81,Z 170.901,A -85,B 0,C 180,E1 -14395.17,E2 -14395.17} C_VEL
LIN {X 0,Y 334.108,Z 170.865,A -85,B 0,C 180,E1 -14397.589,E2 -14397.589} C_VEL
LIN {X 0,Y 334.247,Z 170.852,A -85,B 0,C 180,E1 -14400.001,E2 -14400.001} C_VEL
LIN {X 0,Y 334.106,Z 170.866,A -85,B 0,C 180,E1 -14402.412,E2 -14402.412} C_VEL
LIN {X 0,Y 334,Z 170.882,A -85,B 0,C 180,E1 -14406.04,E2 -14406.04} C_VEL
LIN {X 0,Y 333.822,Z 170.904,A -85,B 0,C 180,E1 -14409.697,E2 -14409.697} C_VEL
LIN {X 0,Y 333.798,Z 170.905,A -85,B 0,C 180,E1 -14413.392,E2 -14413.392} C_VEL
LIN {X 0,Y 333.749,Z 170.91,A -85,B 0,C 180,E1 -14417.147,E2 -14417.147} C_VEL
LIN {X 0,Y 333.741,Z 170.915,A -85,B 0,C 180,E1 -14419.691,E2 -14419.691} C_VEL
LIN {X 0,Y 333.694,Z 170.916,A -85,B 0,C 180,E1 -14422.279,E2 -14422.279} C_VEL
LIN {X 0,Y 333.737,Z 170.91,A -85,B 0,C 180,E1 -14426.247,E2 -14426.247} C_VEL
LIN {X 0,Y 333.692,Z 170.918,A -85,B 0,C 180,E1 -14428.975,E2 -14428.975} C_VEL
LIN {X 0,Y 333.645,Z 170.922,A -85,B 0,C 180,E1 -14432.587,E2 -14432.587} C_VEL
LIN {X 0,Y 333.678,Z 170.918,A -85,B 0,C 180,E1 -14436.139,E2 -14436.139} C_VEL
LIN {X 0,Y 333.649,Z 170.927,A -85,B 0,C 180,E1 -14439.193,E2 -14439.193} C_VEL
LIN {X 0,Y 333.702,Z 171.068,A -85,B 0,C 180,E1 -14442.373,E2 -14442.373} C_VEL
LIN {X 0,Y 334.689,Z 176.478,A -85,B 0,C 180,E1 -14446.136,E2 -14446.136} C_VEL
LIN {X 0,Y 335.667,Z 181.68,A -85,B 0,C 180,E1 -14449.529,E2 -14449.529} C_VEL
LIN {X 0,Y 336.377,Z 186.558,A -85,B 0,C 180,E1 -14452.556,E2 -14452.556} C_VEL
LIN {X 0,Y 336.243,Z 190.104,A -85,B 0,C 180,E1 -14454.604,E2 -14454.604} C_VEL
LIN {X 0,Y 335.534,Z 195.7,A -85,B 0,C 180,E1 -14457.716,E2 -14457.716} C_VEL
LIN {X 0,Y 334.55,Z 203.53,A -85,B 0,C 180,E1 -14461.923,E2 -14461.923} C_VEL
LIN {X 0,Y 333.777,Z 210.864,A -85,B 0,C 180,E1 -14465.758,E2 -14465.758} C_VEL
LIN {X 0,Y 333.336,Z 216.19,A -85,B 0,C 180,E1 -14468.482,E2 -14468.482} C_VEL
LIN {X 0,Y 335.708,Z 230.313,A -85,B 0,C 180,E1 -14469.186,E2 -14469.186} C_VEL
LIN {X 0,Y 337.548,Z 243.946,A -85,B 0,C 180,E1 -14470.118,E2 -14470.118} C_VEL
LIN {X 0,Y 338.751,Z 256.842,A -85,B 0,C 180,E1 -14471.242,E2 -14471.242} C_VEL
LIN {X 0,Y 337.627,Z 267.094,A -85,B 0,C 180,E1 -14472.276,E2 -14472.276} C_VEL
LIN {X 0,Y 336.413,Z 277.759,A -85,B 0,C 180,E1 -14473.619,E2 -14473.619} C_VEL
LIN {X 0,Y 335.399,Z 287.455,A -85,B 0,C 180,E1 -14475.135,E2 -14475.135} C_VEL
LIN {X 0,Y 334.419,Z 295.32,A -85,B 0,C 180,E1 -14476.634,E2 -14476.634} C_VEL
LIN {X 0,Y 333.421,Z 303.054,A -85,B 0,C 180,E1 -14478.449,E2 -14478.449} C_VEL
LIN {X 0,Y 332.82,Z 309.275,A -85,B 0,C 180,E1 -14480.274,E2 -14480.274} C_VEL
LIN {X 0,Y 332.374,Z 314.206,A -85,B 0,C 180,E1 -14482.1,E2 -14482.1} C_VEL
LIN {X 0,Y 332.183,Z 318,A -85,B 0,C 180,E1 -14483.928,E2 -14483.928} C_VEL
LIN {X 0,Y 332.116,Z 319.949,A -85,B 0,C 180,E1 -14485.145,E2 -14485.145} C_VEL
LIN {X 0,Y 332.051,Z 321.469,A -85,B 0,C 180,E1 -14486.36,E2 -14486.36} C_VEL
LIN {X 0,Y 332.129,Z 323.188,A -85,B 0,C 180,E1 -14488.788,E2 -14488.788} C_VEL
LIN {X 0,Y 332.207,Z 323.45,A -85,B 0,C 180,E1 -14490,E2 -14490} C_VEL
LIN {X 0,Y 332.124,Z 323.303,A -85,B 0,C 180,E1 -14491.213,E2 -14491.213} C_VEL
LIN {X 0,Y 332.052,Z 321.727,A -85,B 0,C 180,E1 -14493.641,E2 -14493.641} C_VEL
LIN {X 0,Y 332.078,Z 320.337,A -85,B 0,C 180,E1 -14494.856,E2 -14494.856} C_VEL
LIN {X 0,Y 332.194,Z 317.426,A -85,B 0,C 180,E1 -14496.682,E2 -14496.682} C_VEL
LIN {X 0,Y 332.494,Z 313.487,A -85,B 0,C 180,E1 -14498.509,E2 -14498.509} C_VEL
LIN {X 0,Y 333.032,Z 308.425,A -85,B 0,C 180,E1 -14500.334,E2 -14500.334} C_VEL
LIN {X 0,Y 333.726,Z 302.092,A -85,B 0,C 180,E1 -14502.157,E2 -14502.157} C_VEL
LIN {X 0,Y 334.862,Z 294.26,A -85,B 0,C 180,E1 -14503.967,E2 -14503.967} C_VEL
LIN {X 0,Y 336.124,Z 284.52,A -85,B 0,C 180,E1 -14505.773,E2 -14505.773} C_VEL
LIN {X 0,Y 337.393,Z 274.536,A -85,B 0,C 180,E1 -14507.268,E2 -14507.268} C_VEL
LIN {X 0,Y 338.871,Z 263.356,A -85,B 0,C 180,E1 -14508.595,E2 -14508.595} C_VEL
LIN {X 0,Y 339.426,Z 257.472,A -85,B 0,C 180,E1 -14509.19,E2 -14509.19} C_VEL
LIN {X 0,Y 338.568,Z 244.963,A -85,B 0,C 180,E1 -14510.366,E2 -14510.366} C_VEL
LIN {X 0,Y 337.105,Z 232.021,A -85,B 0,C 180,E1 -14511.34,E2 -14511.34} C_VEL
LIN {X 0,Y 334.552,Z 219.381,A -85,B 0,C 180,E1 -14512.149,E2 -14512.149} C_VEL
LIN {X 0,Y 333.435,Z 214.364,A -85,B 0,C 180,E1 -14512.429,E2 -14512.429} C_VEL
LIN {X 0,Y 334.126,Z 207.141,A -85,B 0,C 180,E1 -14516.214,E2 -14516.214} C_VEL
LIN {X 0,Y 335.052,Z 199.794,A -85,B 0,C 180,E1 -14520.227,E2 -14520.227} C_VEL
LIN {X 0,Y 336.129,Z 192.617,A -85,B 0,C 180,E1 -14524.37,E2 -14524.37} C_VEL
LIN {X 0,Y 336.571,Z 189.115,A -85,B 0,C 180,E1 -14526.521,E2 -14526.521} C_VEL
LIN {X 0,Y 336.352,Z 185.669,A -85,B 0,C 180,E1 -14528.818,E2 -14528.818} C_VEL
LIN {X 0,Y 335.552,Z 181.229,A -85,B 0,C 180,E1 -14532.085,E2 -14532.085} C_VEL
LIN {X 0,Y 334.75,Z 176.974,A -85,B 0,C 180,E1 -14535.547,E2 -14535.547} C_VEL
LIN {X 0,Y 334.031,Z 173.018,A -85,B 0,C 180,E1 -14539.24,E2 -14539.24} C_VEL
LIN {X 0,Y 333.676,Z 170.926,A -85,B 0,C 180,E1 -14541.478,E2 -14541.478} C_VEL
LIN {X 0,Y 333.678,Z 170.92,A -85,B 0,C 180,E1 -14545.341,E2 -14545.341} C_VEL
LIN {X 0,Y 333.694,Z 170.918,A -85,B 0,C 180,E1 -14549.637,E2 -14549.637} C_VEL
LIN {X 0,Y 333.745,Z 170.914,A -85,B 0,C 180,E1 -14552.401,E2 -14552.401} C_VEL
LIN {X 0,Y 333.731,Z 170.912,A -85,B 0,C 180,E1 -14555.09,E2 -14555.09} C_VEL
LIN {X 0,Y 333.684,Z 170.921,A -85,B 0,C 180,E1 -14559.019,E2 -14559.019} C_VEL
LIN {X 0,Y 333.745,Z 170.91,A -85,B 0,C 180,E1 -14561.586,E2 -14561.586} C_VEL
LIN {X 0,Y 333.812,Z 170.906,A -85,B 0,C 180,E1 -14565.576,E2 -14565.576} C_VEL
LIN {X 0,Y 333.838,Z 170.903,A -85,B 0,C 180,E1 -14569.078,E2 -14569.078} C_VEL
LIN {X 0,Y 334.03,Z 170.878,A -85,B 0,C 180,E1 -14572.747,E2 -14572.747} C_VEL
LIN {X 0,Y 333.815,Z 170.905,A -85,B 0,C 180,E1 -14575.169,E2 -14575.169} C_VEL
LIN {X 0,Y 334.111,Z 170.866,A -85,B 0,C 180,E1 -14577.588,E2 -14577.588} C_VEL
LIN {X 0,Y 334.27,Z 170.849,A -85,B 0,C 180,E1 -14579.999,E2 -14579.999} C_VEL
LIN {X 0,Y 334.11,Z 170.867,A -85,B 0,C 180,E1 -14582.411,E2 -14582.411} C_VEL
LIN {X 0,Y 334.002,Z 170.942,A -85,B 0,C 180,E1 -14586.603,E2 -14586.603} C_VEL
LIN {X 0,Y 334.028,Z 171.009,A -85,B 0,C 180,E1 -14587.252,E2 -14587.252} C_VEL
LIN {X 0,Y 333.919,Z 173.509,A -85,B 0,C 180,E1 -14590.918,E2 -14590.918} C_VEL
LIN {X 0,Y 333.676,Z 176.24,A -85,B 0,C 180,E1 -14594.639,E2 -14594.639} C_VEL
LIN {X 0,Y 333.393,Z 179.176,A -85,B 0,C 180,E1 -14598.447,E2 -14598.447} C_VEL
LIN {X 0,Y 333.098,Z 182.537,A -85,B 0,C 180,E1 -14602.605,E2 -14602.605} C_VEL
LIN {X 0,Y 337.981,Z 196.881,A -85,B 0,C 180,E1 -14603.741,E2 -14603.741} C_VEL
LIN {X 0,Y 341.107,Z 208.841,A -85,B 0,C 180,E1 -14604.821,E2 -14604.821} C_VEL
LIN {X 0,Y 341.848,Z 213.019,A -85,B 0,C 180,E1 -14605.231,E2 -14605.231} C_VEL
LIN {X 0,Y 340.686,Z 224.858,A -85,B 0,C 180,E1 -14606.328,E2 -14606.328} C_VEL
LIN {X 0,Y 339.356,Z 235.775,A -85,B 0,C 180,E1 -14607.607,E2 -14607.607} C_VEL
LIN {X 0,Y 337.978,Z 246.246,A -85,B 0,C 180,E1 -14609.148,E2 -14609.148} C_VEL
LIN {X 0,Y 336.668,Z 255.296,A -85,B 0,C 180,E1 -14610.822,E2 -14610.822} C_VEL
LIN {X 0,Y 335.434,Z 263.156,A -85,B 0,C 180,E1 -14612.625,E2 -14612.625} C_VEL
LIN {X 0,Y 334.357,Z 269.851,A -85,B 0,C 180,E1 -14614.577,E2 -14614.577} C_VEL
LIN {X 0,Y 333.512,Z 275.626,A -85,B 0,C 180,E1 -14616.796,E2 -14616.796} C_VEL
LIN {X 0,Y 332.908,Z 279.173,A -85,B 0,C 180,E1 -14618.638,E2 -14618.638} C_VEL
LIN {X 0,Y 332.423,Z 282.162,A -85,B 0,C 180,E1 -14620.949,E2 -14620.949} C_VEL
LIN {X 0,Y 332.16,Z 283.38,A -85,B 0,C 180,E1 -14622.614,E2 -14622.614} C_VEL
LIN {X 0,Y 332.042,Z 283.807,A -85,B 0,C 180,E1 -14624.304,E2 -14624.304} C_VEL
LIN {X 0,Y 332.015,Z 283.457,A -85,B 0,C 180,E1 -14626.029,E2 -14626.029} C_VEL
LIN {X 0,Y 332.122,Z 282.268,A -85,B 0,C 180,E1 -14627.784,E2 -14627.784} C_VEL
LIN {X 0,Y 332.449,Z 280.188,A -85,B 0,C 180,E1 -14629.555,E2 -14629.555} C_VEL
LIN {X 0,Y 332.779,Z 277.059,A -85,B 0,C 180,E1 -14631.389,E2 -14631.389} C_VEL
LIN {X 0,Y 333.241,Z 272.729,A -85,B 0,C 180,E1 -14633.264,E2 -14633.264} C_VEL
LIN {X 0,Y 333.936,Z 266.344,A -85,B 0,C 180,E1 -14635.372,E2 -14635.372} C_VEL
LIN {X 0,Y 334.752,Z 259.642,A -85,B 0,C 180,E1 -14637.116,E2 -14637.116} C_VEL
LIN {X 0,Y 335.738,Z 251.708,A -85,B 0,C 180,E1 -14638.79,E2 -14638.79} C_VEL
LIN {X 0,Y 336.75,Z 242.386,A -85,B 0,C 180,E1 -14640.382,E2 -14640.382} C_VEL
LIN {X 0,Y 337.907,Z 231.149,A -85,B 0,C 180,E1 -14641.928,E2 -14641.928} C_VEL
LIN {X 0,Y 339.028,Z 219.329,A -85,B 0,C 180,E1 -14643.199,E2 -14643.199} C_VEL
LIN {X 0,Y 339.826,Z 210.933,A -85,B 0,C 180,E1 -14643.928,E2 -14643.928} C_VEL
LIN {X 0,Y 338.885,Z 204.301,A -85,B 0,C 180,E1 -14644.491,E2 -14644.491} C_VEL
LIN {X 0,Y 335.819,Z 191.172,A -85,B 0,C 180,E1 -14645.474,E2 -14645.474} C_VEL
LIN {X 0,Y 332.726,Z 179.742,A -85,B 0,C 180,E1 -14646.144,E2 -14646.144} C_VEL
LIN {X 0,Y 332.801,Z 175.882,A -85,B 0,C 180,E1 -14650.252,E2 -14650.252} C_VEL
LIN {X 0,Y 332.998,Z 172.365,A -85,B 0,C 180,E1 -14654.075,E2 -14654.075} C_VEL
LIN {X 0,Y 333.09,Z 171.237,A -85,B 0,C 180,E1 -14655.333,E2 -14655.333} C_VEL
LIN {X 0,Y 333.386,Z 170.956,A -85,B 0,C 180,E1 -14657.83,E2 -14657.83} C_VEL
LIN {X 0,Y 333.918,Z 170.888,A -85,B 0,C 180,E1 -14661.571,E2 -14661.571} C_VEL
LIN {X 0,Y 334.004,Z 170.881,A -85,B 0,C 180,E1 -14663.961,E2 -14663.961} C_VEL
LIN {X 0,Y 334.104,Z 170.866,A -85,B 0,C 180,E1 -14667.589,E2 -14667.589} C_VEL
LIN {X 0,Y 334.263,Z 170.85,A -85,B 0,C 180,E1 -14670,E2 -14670} C_VEL
LIN {X 0,Y 334.104,Z 170.866,A -85,B 0,C 180,E1 -14672.411,E2 -14672.411} C_VEL
LIN {X 0,Y 334.021,Z 170.876,A -85,B 0,C 180,E1 -14677.252,E2 -14677.252} C_VEL
LIN {X 0,Y 333.83,Z 170.899,A -85,B 0,C 180,E1 -14680.922,E2 -14680.922} C_VEL
LIN {X 0,Y 333.805,Z 170.902,A -85,B 0,C 180,E1 -14684.634,E2 -14684.634} C_VEL
LIN {X 0,Y 333.792,Z 170.903,A -85,B 0,C 180,E1 -14688.655,E2 -14688.655} C_VEL
LIN {X 0,Y 333.689,Z 170.917,A -85,B 0,C 180,E1 -14692.278,E2 -14692.278} C_VEL
LIN {X 0,Y 333.732,Z 170.911,A -85,B 0,C 180,E1 -14696.246,E2 -14696.246} C_VEL
LIN {X 0,Y 333.686,Z 170.919,A -85,B 0,C 180,E1 -14698.974,E2 -14698.974} C_VEL
LIN {X 0,Y 333.64,Z 170.923,A -85,B 0,C 180,E1 -14702.587,E2 -14702.587} C_VEL
LIN {X 0,Y 333.673,Z 170.918,A -85,B 0,C 180,E1 -14706.139,E2 -14706.139} C_VEL
LIN {X 0,Y 333.643,Z 170.928,A -85,B 0,C 180,E1 -14709.193,E2 -14709.193} C_VEL
LIN {X 0,Y 333.63,Z 170.925,A -85,B 0,C 180,E1 -14712.501,E2 -14712.501} C_VEL
LIN {X 0,Y 333.618,Z 170.925,A -85,B 0,C 180,E1 -14715.96,E2 -14715.96} C_VEL
LIN {X 0,Y 333.645,Z 170.924,A -85,B 0,C 180,E1 -14719.316,E2 -14719.316} C_VEL
LIN {X 0,Y 333.663,Z 170.922,A -85,B 0,C 180,E1 -14723.168,E2 -14723.168} C_VEL
LIN {X 0,Y 333.637,Z 170.923,A -85,B 0,C 180,E1 -14725.803,E2 -14725.803} C_VEL
LIN {X 0,Y 332.942,Z 171.015,A -85,B 0,C 180,E1 -14726.811,E2 -14726.811} C_VEL
LIN {X 0,Y 330.095,Z 171.367,A -85,B 0,C 180,E1 -14728.452,E2 -14728.452} C_VEL
LIN {X 0,Y 327.709,Z 171.661,A -85,B 0,C 180,E1 -14729.781,E2 -14729.781} C_VEL
LIN {X 0,Y 326.699,Z 171.791,A -85,B 0,C 180,E1 -14730.81,E2 -14730.81} C_VEL
LIN {X 0,Y 326.623,Z 171.794,A -85,B 0,C 180,E1 -14731.158,E2 -14731.158} C_VEL
LIN {X 0,Y 326.687,Z 171.794,A -85,B 0,C 180,E1 -14734.628,E2 -14734.628} C_VEL
LIN {X 0,Y 326.648,Z 171.799,A -85,B 0,C 180,E1 -14738.546,E2 -14738.546} C_VEL
LIN {X 0,Y 326.744,Z 171.782,A -85,B 0,C 180,E1 -14741.178,E2 -14741.178} C_VEL
LIN {X 0,Y 326.763,Z 171.779,A -85,B 0,C 180,E1 -14745.434,E2 -14745.434} C_VEL
LIN {X 0,Y 326.77,Z 171.779,A -85,B 0,C 180,E1 -14748.84,E2 -14748.84} C_VEL
LIN {X 0,Y 326.957,Z 171.757,A -85,B 0,C 180,E1 -14752.591,E2 -14752.591} C_VEL
LIN {X 0,Y 326.777,Z 171.777,A -85,B 0,C 180,E1 -14755.066,E2 -14755.066} C_VEL
LIN {X 0,Y 327.049,Z 171.744,A -85,B 0,C 180,E1 -14757.537,E2 -14757.537} C_VEL
LIN {X 0,Y 327.198,Z 171.73,A -85,B 0,C 180,E1 -14760.001,E2 -14760.001} C_VEL
LIN {X 0,Y 327.047,Z 171.745,A -85,B 0,C 180,E1 -14762.464,E2 -14762.464} C_VEL
LIN {X 0,Y 326.954,Z 171.758,A -85,B 0,C 180,E1 -14766.171,E2 -14766.171} C_VEL
LIN {X 0,Y 326.785,Z 171.781,A -85,B 0,C 180,E1 -14769.908,E2 -14769.908} C_VEL
LIN {X 0,Y 326.761,Z 171.784,A -85,B 0,C 180,E1 -14773.686,E2 -14773.686} C_VEL
LIN {X 0,Y 326.702,Z 171.791,A -85,B 0,C 180,E1 -14777.528,E2 -14777.528} C_VEL
LIN {X 0,Y 326.667,Z 171.792,A -85,B 0,C 180,E1 -14780.135,E2 -14780.135} C_VEL
LIN {X 0,Y 326.654,Z 171.793,A -85,B 0,C 180,E1 -14784.129,E2 -14784.129} C_VEL
LIN {X 0,Y 326.685,Z 171.79,A -85,B 0,C 180,E1 -14786.858,E2 -14786.858} C_VEL
LIN {X 0,Y 326.636,Z 171.795,A -85,B 0,C 180,E1 -14790.61,E2 -14790.61} C_VEL
LIN {X 0,Y 326.609,Z 171.799,A -85,B 0,C 180,E1 -14794.02,E2 -14794.02} C_VEL
LIN {X 0,Y 326.629,Z 171.801,A -85,B 0,C 180,E1 -14797.239,E2 -14797.239} C_VEL
LIN {X 0,Y 326.602,Z 171.805,A -85,B 0,C 180,E1 -14801.136,E2 -14801.136} C_VEL
LIN {X 0,Y 326.694,Z 172.009,A -85,B 0,C 180,E1 -14802.035,E2 -14802.035} C_VEL
LIN {X 0,Y 327.658,Z 177.446,A -85,B 0,C 180,E1 -14805.888,E2 -14805.888} C_VEL
LIN {X 0,Y 328.608,Z 182.559,A -85,B 0,C 180,E1 -14809.322,E2 -14809.322} C_VEL
LIN {X 0,Y 329.289,Z 187.025,A -85,B 0,C 180,E1 -14812.157,E2 -14812.157} C_VEL
LIN {X 0,Y 329.288,Z 190.451,A -85,B 0,C 180,E1 -14814.198,E2 -14814.198} C_VEL
LIN {X 0,Y 328.488,Z 196.53,A -85,B 0,C 180,E1 -14817.665,E2 -14817.665} C_VEL
LIN {X 0,Y 327.495,Z 204.11,A -85,B 0,C 180,E1 -14821.828,E2 -14821.828} C_VEL
LIN {X 0,Y 326.812,Z 210.386,A -85,B 0,C 180,E1 -14825.207,E2 -14825.207} C_VEL
LIN {X 0,Y 326.319,Z 215.932,A -85,B 0,C 180,E1 -14828.069,E2 -14828.069} C_VEL
LIN {X 0,Y 328.685,Z 229.811,A -85,B 0,C 180,E1 -14828.772,E2 -14828.772} C_VEL
LIN {X 0,Y 330.43,Z 242.41,A -85,B 0,C 180,E1 -14829.644,E2 -14829.644} C_VEL
LIN {X 0,Y 331.493,Z 254.098,A -85,B 0,C 180,E1 -14830.655,E2 -14830.655} C_VEL
LIN {X 0,Y 331.775,Z 259.087,A -85,B 0,C 180,E1 -14831.153,E2 -14831.153} C_VEL
LIN {X 0,Y 330.404,Z 270.133,A -85,B 0,C 180,E1 -14832.356,E2 -14832.356} C_VEL
LIN {X 0,Y 329.324,Z 279.141,A -85,B 0,C 180,E1 -14833.575,E2 -14833.575} C_VEL
LIN {X 0,Y 328.281,Z 288.429,A -85,B 0,C 180,E1 -14835.114,E2 -14835.114} C_VEL
LIN {X 0,Y 327.066,Z 297.439,A -85,B 0,C 180,E1 -14836.961,E2 -14836.961} C_VEL
LIN {X 0,Y 326.16,Z 304.709,A -85,B 0,C 180,E1 -14838.818,E2 -14838.818} C_VEL
LIN {X 0,Y 325.608,Z 310.528,A -85,B 0,C 180,E1 -14840.684,E2 -14840.684} C_VEL
LIN {X 0,Y 325.207,Z 315.095,A -85,B 0,C 180,E1 -14842.55,E2 -14842.55} C_VEL
LIN {X 0,Y 325.104,Z 317.758,A -85,B 0,C 180,E1 -14843.945,E2 -14843.945} C_VEL
LIN {X 0,Y 324.981,Z 320.999,A -85,B 0,C 180,E1 -14846.28,E2 -14846.28} C_VEL
LIN {X 0,Y 324.95,Z 322.078,A -85,B 0,C 180,E1 -14847.521,E2 -14847.521} C_VEL
LIN {X 0,Y 325.037,Z 322.748,A -85,B 0,C 180,E1 -14848.761,E2 -14848.761} C_VEL
LIN {X 0,Y 325.132,Z 323.021,A -85,B 0,C 180,E1 -14850,E2 -14850} C_VEL
LIN {X 0,Y 325.03,Z 322.887,A -85,B 0,C 180,E1 -14851.239,E2 -14851.239} C_VEL
LIN {X 0,Y 324.939,Z 322.316,A -85,B 0,C 180,E1 -14852.479,E2 -14852.479} C_VEL
LIN {X 0,Y 324.979,Z 321.338,A -85,B 0,C 180,E1 -14853.72,E2 -14853.72} C_VEL
LIN {X 0,Y 325.111,Z 318.167,A -85,B 0,C 180,E1 -14856.205,E2 -14856.205} C_VEL
LIN {X 0,Y 325.302,Z 314.602,A -85,B 0,C 180,E1 -14858.073,E2 -14858.073} C_VEL
LIN {X 0,Y 325.805,Z 309.966,A -85,B 0,C 180,E1 -14859.938,E2 -14859.938} C_VEL
LIN {X 0,Y 326.615,Z 302.988,A -85,B 0,C 180,E1 -14862.111,E2 -14862.111} C_VEL
LIN {X 0,Y 327.748,Z 295.477,A -85,B 0,C 180,E1 -14863.96,E2 -14863.96} C_VEL
LIN {X 0,Y 328.939,Z 287.005,A -85,B 0,C 180,E1 -14865.657,E2 -14865.657} C_VEL
LIN {X 0,Y 330.291,Z 276.618,A -85,B 0,C 180,E1 -14867.331,E2 -14867.331} C_VEL
LIN {X 0,Y 331.79,Z 266.095,A -85,B 0,C 180,E1 -14868.686,E2 -14868.686} C_VEL
LIN {X 0,Y 332.663,Z 259.163,A -85,B 0,C 180,E1 -14869.436,E2 -14869.436} C_VEL
LIN {X 0,Y 331.872,Z 245.65,A -85,B 0,C 180,E1 -14870.767,E2 -14870.767} C_VEL
LIN {X 0,Y 330.454,Z 232.714,A -85,B 0,C 180,E1 -14871.807,E2 -14871.807} C_VEL
LIN {X 0,Y 327.922,Z 220.035,A -85,B 0,C 180,E1 -14872.664,E2 -14872.664} C_VEL
LIN {X 0,Y 326.454,Z 213.893,A -85,B 0,C 180,E1 -14873.026,E2 -14873.026} C_VEL
LIN {X 0,Y 327.18,Z 206.892,A -85,B 0,C 180,E1 -14876.814,E2 -14876.814} C_VEL
LIN {X 0,Y 328,Z 200.801,A -85,B 0,C 180,E1 -14880.234,E2 -14880.234} C_VEL
LIN {X 0,Y 328.93,Z 194.841,A -85,B 0,C 180,E1 -14883.747,E2 -14883.747} C_VEL
LIN {X 0,Y 329.593,Z 190.159,A -85,B 0,C 180,E1 -14886.659,E2 -14886.659} C_VEL
LIN {X 0,Y 329.363,Z 186.79,A -85,B 0,C 180,E1 -14888.978,E2 -14888.978} C_VEL
LIN {X 0,Y 328.537,Z 182.303,A -85,B 0,C 180,E1 -14892.364,E2 -14892.364} C_VEL
LIN {X 0,Y 327.62,Z 177.311,A -85,B 0,C 180,E1 -14896.649,E2 -14896.649} C_VEL
LIN {X 0,Y 326.871,Z 173.243,A -85,B 0,C 180,E1 -14900.718,E2 -14900.718} C_VEL
LIN {X 0,Y 326.609,Z 171.803,A -85,B 0,C 180,E1 -14902.502,E2 -14902.502} C_VEL
LIN {X 0,Y 326.611,Z 171.801,A -85,B 0,C 180,E1 -14905.98,E2 -14905.98} C_VEL
LIN {X 0,Y 326.652,Z 171.798,A -85,B 0,C 180,E1 -14910.339,E2 -14910.339} C_VEL
LIN {X 0,Y 326.694,Z 171.792,A -85,B 0,C 180,E1 -14914.516,E2 -14914.516} C_VEL
LIN {X 0,Y 326.65,Z 171.799,A -85,B 0,C 180,E1 -14918.545,E2 -14918.545} C_VEL
LIN {X 0,Y 326.711,Z 171.789,A -85,B 0,C 180,E1 -14921.175,E2 -14921.175} C_VEL
LIN {X 0,Y 326.767,Z 171.783,A -85,B 0,C 180,E1 -14925.433,E2 -14925.433} C_VEL
LIN {X 0,Y 326.774,Z 171.783,A -85,B 0,C 180,E1 -14928.838,E2 -14928.838} C_VEL
LIN {X 0,Y 326.984,Z 171.757,A -85,B 0,C 180,E1 -14932.59,E2 -14932.59} C_VEL
LIN {X 0,Y 326.782,Z 171.781,A -85,B 0,C 180,E1 -14935.064,E2 -14935.064} C_VEL
LIN {X 0,Y 327.052,Z 171.745,A -85,B 0,C 180,E1 -14937.536,E2 -14937.536} C_VEL
LIN {X 0,Y 327.221,Z 171.727,A -85,B 0,C 180,E1 -14939.999,E2 -14939.999} C_VEL
LIN {X 0,Y 327.051,Z 171.747,A -85,B 0,C 180,E1 -14942.463,E2 -14942.463} C_VEL
LIN {X 0,Y 326.973,Z 171.761,A -85,B 0,C 180,E1 -14946.169,E2 -14946.169} C_VEL
LIN {X 0,Y 327.011,Z 173.164,A -85,B 0,C 180,E1 -14948.652,E2 -14948.652} C_VEL
LIN {X 0,Y 326.807,Z 175.757,A -85,B 0,C 180,E1 -14952.418,E2 -14952.418} C_VEL
LIN {X 0,Y 326.618,Z 177.609,A -85,B 0,C 180,E1 -14954.963,E2 -14954.963} C_VEL
LIN {X 0,Y 326.32,Z 180.553,A -85,B 0,C 180,E1 -14958.847,E2 -14958.847} C_VEL
LIN {X 0,Y 326.155,Z 183.252,A -85,B 0,C 180,E1 -14962.043,E2 -14962.043} C_VEL
LIN {X 0,Y 330.863,Z 196.692,A -85,B 0,C 180,E1 -14963.138,E2 -14963.138} C_VEL
LIN {X 0,Y 334.029,Z 208.379,A -85,B 0,C 180,E1 -14964.221,E2 -14964.221} C_VEL
LIN {X 0,Y 335.218,Z 213.925,A -85,B 0,C 180,E1 -14964.79,E2 -14964.79} C_VEL
LIN {X 0,Y 334.105,Z 225.373,A -85,B 0,C 180,E1 -14965.885,E2 -14965.885} C_VEL
LIN {X 0,Y 332.755,Z 235.851,A -85,B 0,C 180,E1 -14967.133,E2 -14967.133} C_VEL
LIN {X 0,Y 331.354,Z 246.214,A -85,B 0,C 180,E1 -14968.676,E2 -14968.676} C_VEL
LIN {X 0,Y 329.941,Z 255.416,A -85,B 0,C 180,E1 -14970.397,E2 -14970.397} C_VEL
LIN {X 0,Y 328.569,Z 263.689,A -85,B 0,C 180,E1 -14972.326,E2 -14972.326} C_VEL
LIN {X 0,Y 327.625,Z 269.096,A -85,B 0,C 180,E1 -14973.898,E2 -14973.898} C_VEL
LIN {X 0,Y 326.944,Z 273.524,A -85,B 0,C 180,E1 -14975.477,E2 -14975.477} C_VEL
LIN {X 0,Y 326.074,Z 278.712,A -85,B 0,C 180,E1 -14977.897,E2 -14977.897} C_VEL
LIN {X 0,Y 325.743,Z 280.515,A -85,B 0,C 180,E1 -14979.039,E2 -14979.039} C_VEL
LIN {X 0,Y 325.372,Z 282.672,A -85,B 0,C 180,E1 -14980.887,E2 -14980.887} C_VEL
LIN {X 0,Y 325.076,Z 283.901,A -85,B 0,C 180,E1 -14982.687,E2 -14982.687} C_VEL
LIN {X 0,Y 324.973,Z 284.259,A -85,B 0,C 180,E1 -14984.465,E2 -14984.465} C_VEL
LIN {X 0,Y 324.945,Z 283.798,A -85,B 0,C 180,E1 -14986.203,E2 -14986.203} C_VEL
LIN {X 0,Y 325.048,Z 282.582,A -85,B 0,C 180,E1 -14987.912,E2 -14987.912} C_VEL
LIN {X 0,Y 325.368,Z 280.604,A -85,B 0,C 180,E1 -14989.608,E2 -14989.608} C_VEL
LIN {X 0,Y 325.689,Z 277.889,A -85,B 0,C 180,E1 -14991.26,E2 -14991.26} C_VEL
LIN {X 0,Y 326.292,Z 272.355,A -85,B 0,C 180,E1 -14993.685,E2 -14993.685} C_VEL
LIN {X 0,Y 327.004,Z 266.087,A -85,B 0,C 180,E1 -14995.741,E2 -14995.741} C_VEL
LIN {X 0,Y 327.921,Z 258.857,A -85,B 0,C 180,E1 -14997.601,E2 -14997.601} C_VEL
LIN {X 0,Y 329.153,Z 249.423,A -85,B 0,C 180,E1 -14999.528,E2 -14999.528} C_VEL
LIN {X 0,Y 330.243,Z 239.715,A -85,B 0,C 180,E1 -15001.122,E2 -15001.122} C_VEL
LIN {X 0,Y 331.381,Z 228.666,A -85,B 0,C 180,E1 -15002.57,E2 -15002.57} C_VEL
LIN {X 0,Y 332.502,Z 216.655,A -85,B 0,C 180,E1 -15003.817,E2 -15003.817} C_VEL
LIN {X 0,Y 332.925,Z 210.319,A -85,B 0,C 180,E1 -15004.357,E2 -15004.357} C_VEL
LIN {X 0,Y 330.572,Z 198.789,A -85,B 0,C 180,E1 -15005.34,E2 -15005.34} C_VEL
LIN {X 0,Y 327.34,Z 186.156,A -85,B 0,C 180,E1 -15006.219,E2 -15006.219} C_VEL
LIN {X 0,Y 325.651,Z 180.105,A -85,B 0,C 180,E1 -15006.594,E2 -15006.594} C_VEL
LIN {X 0,Y 325.735,Z 177.111,A -85,B 0,C 180,E1 -15009.805,E2 -15009.805} C_VEL
LIN {X 0,Y 325.926,Z 173.553,A -85,B 0,C 180,E1 -15013.72,E2 -15013.72} C_VEL
LIN {X 0,Y 326.124,Z 171.863,A -85,B 0,C 180,E1 -15015.869,E2 -15015.869} C_VEL
LIN {X 0,Y 326.635,Z 171.799,A -85,B 0,C 180,E1 -15020.088,E2 -15020.088} C_VEL
LIN {X 0,Y 326.935,Z 171.76,A -85,B 0,C 180,E1 -15022.589,E2 -15022.589} C_VEL
LIN {X 0,Y 326.978,Z 171.755,A -85,B 0,C 180,E1 -15023.83,E2 -15023.83} C_VEL
LIN {X 0,Y 327.044,Z 171.745,A -85,B 0,C 180,E1 -15027.537,E2 -15027.537} C_VEL
LIN {X 0,Y 327.214,Z 171.728,A -85,B 0,C 180,E1 -15030,E2 -15030} C_VEL
LIN {X 0,Y 327.045,Z 171.745,A -85,B 0,C 180,E1 -15032.463,E2 -15032.463} C_VEL
LIN {X 0,Y 326.992,Z 171.753,A -85,B 0,C 180,E1 -15036.169,E2 -15036.169} C_VEL
LIN {X 0,Y 326.911,Z 171.761,A -85,B 0,C 180,E1 -15038.655,E2 -15038.655} C_VEL
LIN {X 0,Y 326.731,Z 171.784,A -85,B 0,C 180,E1 -15042.421,E2 -15042.421} C_VEL
LIN {X 0,Y 326.751,Z 171.781,A -85,B 0,C 180,E1 -15044.957,E2 -15044.957} C_VEL
LIN {X 0,Y 326.729,Z 171.783,A -85,B 0,C 180,E1 -15048.838,E2 -15048.838} C_VEL
LIN {X 0,Y 326.618,Z 171.797,A -85,B 0,C 180,E1 -15052.787,E2 -15052.787} C_VEL
LIN {X 0,Y 326.686,Z 171.794,A -85,B 0,C 180,E1 -15055.484,E2 -15055.484} C_VEL
LIN {X 0,Y 326.644,Z 171.797,A -85,B 0,C 180,E1 -15059.661,E2 -15059.661} C_VEL
LIN {X 0,Y 326.603,Z 171.799,A -85,B 0,C 180,E1 -15064.02,E2 -15064.02} C_VEL
LIN {X 0,Y 326.624,Z 171.802,A -85,B 0,C 180,E1 -15067.239,E2 -15067.239} C_VEL
LIN {X 0,Y 326.575,Z 171.808,A -85,B 0,C 180,E1 -15071.132,E2 -15071.132} C_VEL
LIN {X 0,Y 326.553,Z 171.808,A -85,B 0,C 180,E1 -15074.748,E2 -15074.748} C_VEL
LIN {X 0,Y 326.574,Z 171.802,A -85,B 0,C 180,E1 -15078.155,E2 -15078.155} C_VEL
LIN {X 0,Y 326.596,Z 171.801,A -85,B 0,C 180,E1 -15081.388,E2 -15081.388} C_VEL
LIN {X 0,Y 326.618,Z 171.802,A -85,B 0,C 180,E1 -15084.852,E2 -15084.852} C_VEL
LIN {X 0,Y 326.606,Z 171.799,A -85,B 0,C 180,E1 -15087.456,E2 -15087.456} C_VEL
LIN {X 0,Y 326.623,Z 171.794,A -85,B 0,C 180,E1 -15091.158,E2 -15091.158} C_VEL
LIN {X 0,Y 325.964,Z 171.881,A -85,B 0,C 180,E1 -15092.188,E2 -15092.188} C_VEL
LIN {X 0,Y 323.088,Z 172.237,A -85,B 0,C 180,E1 -15093.863,E2 -15093.863} C_VEL
LIN {X 0,Y 320.658,Z 172.54,A -85,B 0,C 180,E1 -15095.221,E2 -15095.221} C_VEL
LIN {X 0,Y 319.638,Z 172.669,A -85,B 0,C 180,E1 -15096.273,E2 -15096.273} C_VEL
LIN {X 0,Y 319.568,Z 172.679,A -85,B 0,C 180,E1 -15096.629,E2 -15096.629} C_VEL
LIN {X 0,Y 319.688,Z 172.661,A -85,B 0,C 180,E1 -15100.963,E2 -15100.963} C_VEL
LIN {X 0,Y 319.731,Z 172.654,A -85,B 0,C 180,E1 -15105.276,E2 -15105.276} C_VEL
LIN {X 0,Y 319.753,Z 172.654,A -85,B 0,C 180,E1 -15109.873,E2 -15109.873} C_VEL
LIN {X 0,Y 319.912,Z 172.636,A -85,B 0,C 180,E1 -15112.426,E2 -15112.426} C_VEL
LIN {X 0,Y 319.746,Z 172.653,A -85,B 0,C 180,E1 -15114.957,E2 -15114.957} C_VEL
LIN {X 0,Y 319.993,Z 172.622,A -85,B 0,C 180,E1 -15117.483,E2 -15117.483} C_VEL
LIN {X 0,Y 320.15,Z 172.607,A -85,B 0,C 180,E1 -15120.001,E2 -15120.001} C_VEL
LIN {X 0,Y 319.99,Z 172.624,A -85,B 0,C 180,E1 -15122.518,E2 -15122.518} C_VEL
LIN {X 0,Y 319.91,Z 172.634,A -85,B 0,C 180,E1 -15126.307,E2 -15126.307} C_VEL
LIN {X 0,Y 319.737,Z 172.657,A -85,B 0,C 180,E1 -15130.128,E2 -15130.128} C_VEL
LIN {X 0,Y 319.734,Z 172.658,A -85,B 0,C 180,E1 -15133.993,E2 -15133.993} C_VEL
LIN {X 0,Y 319.661,Z 172.666,A -85,B 0,C 180,E1 -15137.927,E2 -15137.927} C_VEL
LIN {X 0,Y 319.617,Z 172.669,A -85,B 0,C 180,E1 -15140.599,E2 -15140.599} C_VEL
LIN {X 0,Y 319.572,Z 172.678,A -85,B 0,C 180,E1 -15143.32,E2 -15143.32} C_VEL
LIN {X 0,Y 319.62,Z 172.67,A -85,B 0,C 180,E1 -15146.09,E2 -15146.09} C_VEL
LIN {X 0,Y 319.582,Z 172.675,A -85,B 0,C 180,E1 -15148.935,E2 -15148.935} C_VEL
LIN {X 0,Y 319.533,Z 172.681,A -85,B 0,C 180,E1 -15151.862,E2 -15151.862} C_VEL
LIN {X 0,Y 319.582,Z 172.677,A -85,B 0,C 180,E1 -15155.544,E2 -15155.544} C_VEL
LIN {X 0,Y 319.559,Z 172.682,A -85,B 0,C 180,E1 -15158.011,E2 -15158.011} C_VEL
LIN {X 0,Y 319.622,Z 172.879,A -85,B 0,C 180,E1 -15161.616,E2 -15161.616} C_VEL
LIN {X 0,Y 320.565,Z 178.116,A -85,B 0,C 180,E1 -15165.448,E2 -15165.448} C_VEL
LIN {X 0,Y 321.55,Z 183.325,A -85,B 0,C 180,E1 -15169.027,E2 -15169.027} C_VEL
LIN {X 0,Y 322.305,Z 188.485,A -85,B 0,C 180,E1 -15172.371,E2 -15172.371} C_VEL
LIN {X 0,Y 322.128,Z 192.295,A -85,B 0,C 180,E1 -15174.679,E2 -15174.679} C_VEL
LIN {X 0,Y 321.455,Z 197.327,A -85,B 0,C 180,E1 -15177.612,E2 -15177.612} C_VEL
LIN {X 0,Y 320.552,Z 203.844,A -85,B 0,C 180,E1 -15181.282,E2 -15181.282} C_VEL
LIN {X 0,Y 319.712,Z 211.169,A -85,B 0,C 180,E1 -15185.313,E2 -15185.313} C_VEL
LIN {X 0,Y 319.281,Z 215.493,A -85,B 0,C 180,E1 -15187.63,E2 -15187.63} C_VEL
LIN {X 0,Y 321.674,Z 229.287,A -85,B 0,C 180,E1 -15188.352,E2 -15188.352} C_VEL
LIN {X 0,Y 323.302,Z 241.227,A -85,B 0,C 180,E1 -15189.188,E2 -15189.188} C_VEL
LIN {X 0,Y 324.477,Z 253.003,A -85,B 0,C 180,E1 -15190.219,E2 -15190.219} C_VEL
LIN {X 0,Y 324.854,Z 259.684,A -85,B 0,C 180,E1 -15190.9,E2 -15190.9} C_VEL
LIN {X 0,Y 323.444,Z 270.514,A -85,B 0,C 180,E1 -15192.127,E2 -15192.127} C_VEL
LIN {X 0,Y 322.217,Z 280.37,A -85,B 0,C 180,E1 -15193.528,E2 -15193.528} C_VEL
LIN {X 0,Y 321.141,Z 289.368,A -85,B 0,C 180,E1 -15195.1,E2 -15195.1} C_VEL
LIN {X 0,Y 319.927,Z 298.155,A -85,B 0,C 180,E1 -15196.987,E2 -15196.987} C_VEL
LIN {X 0,Y 319.046,Z 305.177,A -85,B 0,C 180,E1 -15198.887,E2 -15198.887} C_VEL
LIN {X 0,Y 318.405,Z 311.613,A -85,B 0,C 180,E1 -15201.112,E2 -15201.112} C_VEL
LIN {X 0,Y 318.073,Z 315.832,A -85,B 0,C 180,E1 -15203.02,E2 -15203.02} C_VEL
LIN {X 0,Y 317.95,Z 318.972,A -85,B 0,C 180,E1 -15204.928,E2 -15204.928} C_VEL
LIN {X 0,Y 317.912,Z 320.525,A -85,B 0,C 180,E1 -15206.198,E2 -15206.198} C_VEL
LIN {X 0,Y 317.866,Z 321.626,A -85,B 0,C 180,E1 -15207.466,E2 -15207.466} C_VEL
LIN {X 0,Y 317.944,Z 322.306,A -85,B 0,C 180,E1 -15208.734,E2 -15208.734} C_VEL
LIN {X 0,Y 318.043,Z 322.591,A -85,B 0,C 180,E1 -15210,E2 -15210} C_VEL
LIN {X 0,Y 317.936,Z 322.468,A -85,B 0,C 180,E1 -15211.267,E2 -15211.267} C_VEL
LIN {X 0,Y 317.856,Z 321.922,A -85,B 0,C 180,E1 -15212.535,E2 -15212.535} C_VEL
LIN {X 0,Y 317.907,Z 320.958,A -85,B 0,C 180,E1 -15213.803,E2 -15213.803} C_VEL
LIN {X 0,Y 318.021,Z 317.818,A -85,B 0,C 180,E1 -15216.344,E2 -15216.344} C_VEL
LIN {X 0,Y 318.242,Z 314.282,A -85,B 0,C 180,E1 -15218.253,E2 -15218.253} C_VEL
LIN {X 0,Y 318.76,Z 309.677,A -85,B 0,C 180,E1 -15220.159,E2 -15220.159} C_VEL
LIN {X 0,Y 319.626,Z 302.754,A -85,B 0,C 180,E1 -15222.38,E2 -15222.38} C_VEL
LIN {X 0,Y 320.834,Z 295.283,A -85,B 0,C 180,E1 -15224.267,E2 -15224.267} C_VEL
LIN {X 0,Y 322.162,Z 286.305,A -85,B 0,C 180,E1 -15226.104,E2 -15226.104} C_VEL
LIN {X 0,Y 323.661,Z 275.519,A -85,B 0,C 180,E1 -15227.861,E2 -15227.861} C_VEL
LIN {X 0,Y 325.284,Z 264.908,A -85,B 0,C 180,E1 -15229.238,E2 -15229.238} C_VEL
LIN {X 0,Y 325.88,Z 259.383,A -85,B 0,C 180,E1 -15229.857,E2 -15229.857} C_VEL
LIN {X 0,Y 325.29,Z 247.744,A -85,B 0,C 180,E1 -15231.068,E2 -15231.068} C_VEL
LIN {X 0,Y 324.087,Z 235.321,A -85,B 0,C 180,E1 -15232.137,E2 -15232.137} C_VEL
LIN {X 0,Y 321.717,Z 222.546,A -85,B 0,C 180,E1 -15233.079,E2 -15233.079} C_VEL
LIN {X 0,Y 319.466,Z 213.363,A -85,B 0,C 180,E1 -15233.684,E2 -15233.684} C_VEL
LIN {X 0,Y 320.284,Z 206.643,A -85,B 0,C 180,E1 -15237.439,E2 -15237.439} C_VEL
LIN {X 0,Y 321.338,Z 199.415,A -85,B 0,C 180,E1 -15241.662,E2 -15241.662} C_VEL
LIN {X 0,Y 322.333,Z 193.541,A -85,B 0,C 180,E1 -15245.296,E2 -15245.296} C_VEL
LIN {X 0,Y 322.547,Z 190.084,A -85,B 0,C 180,E1 -15247.597,E2 -15247.597} C_VEL
LIN {X 0,Y 322.086,Z 186.506,A -85,B 0,C 180,E1 -15250.207,E2 -15250.207} C_VEL
LIN {X 0,Y 321.261,Z 182.087,A -85,B 0,C 180,E1 -15253.786,E2 -15253.786} C_VEL
LIN {X 0,Y 320.575,Z 178.31,A -85,B 0,C 180,E1 -15257.186,E2 -15257.186} C_VEL
LIN {X 0,Y 320.015,Z 175.141,A -85,B 0,C 180,E1 -15260.44,E2 -15260.44} C_VEL
LIN {X 0,Y 319.563,Z 172.68,A -85,B 0,C 180,E1 -15263.572,E2 -15263.572} C_VEL
LIN {X 0,Y 319.581,Z 172.678,A -85,B 0,C 180,E1 -15266.686,E2 -15266.686} C_VEL
LIN {X 0,Y 319.589,Z 172.675,A -85,B 0,C 180,E1 -15269.616,E2 -15269.616} C_VEL
LIN {X 0,Y 319.61,Z 172.674,A -85,B 0,C 180,E1 -15272.498,E2 -15272.498} C_VEL
LIN {X 0,Y 319.609,Z 172.671,A -85,B 0,C 180,E1 -15275.304,E2 -15275.304} C_VEL
LIN {X 0,Y 319.601,Z 172.674,A -85,B 0,C 180,E1 -15278.047,E2 -15278.047} C_VEL
LIN {X 0,Y 319.661,Z 172.668,A -85,B 0,C 180,E1 -15280.978,E2 -15280.978} C_VEL
LIN {X 0,Y 319.716,Z 172.661,A -85,B 0,C 180,E1 -15285.288,E2 -15285.288} C_VEL
LIN {X 0,Y 319.727,Z 172.66,A -85,B 0,C 180,E1 -15288.589,E2 -15288.589} C_VEL
LIN {X 0,Y 319.937,Z 172.634,A -85,B 0,C 180,E1 -15292.426,E2 -15292.426} C_VEL
LIN {X 0,Y 319.752,Z 172.657,A -85,B 0,C 180,E1 -15294.956,E2 -15294.956} C_VEL
LIN {X 0,Y 319.996,Z 172.624,A -85,B 0,C 180,E1 -15297.482,E2 -15297.482} C_VEL
LIN {X 0,Y 320.172,Z 172.605,A -85,B 0,C 180,E1 -15299.999,E2 -15299.999} C_VEL
LIN {X 0,Y 319.995,Z 172.626,A -85,B 0,C 180,E1 -15302.517,E2 -15302.517} C_VEL
LIN {X 0,Y 319.747,Z 172.659,A -85,B 0,C 180,E1 -15305.043,E2 -15305.043} C_VEL
LIN {X 0,Y 319.976,Z 173.163,A -85,B 0,C 180,E1 -15306.622,E2 -15306.622} C_VEL
LIN {X 0,Y 320.015,Z 174.538,A -85,B 0,C 180,E1 -15308.842,E2 -15308.842} C_VEL
LIN {X 0,Y 319.791,Z 177.115,A -85,B 0,C 180,E1 -15312.695,E2 -15312.695} C_VEL
LIN {X 0,Y 319.568,Z 178.972,A -85,B 0,C 180,E1 -15315.301,E2 -15315.301} C_VEL
LIN {X 0,Y 319.249,Z 181.941,A -85,B 0,C 180,E1 -15319.281,E2 -15319.281} C_VEL
LIN {X 0,Y 319.153,Z 183.571,A -85,B 0,C 180,E1 -15321.39,E2 -15321.39} C_VEL
LIN {X 0,Y 321.266,Z 189.453,A -85,B 0,C 180,E1 -15321.862,E2 -15321.862} C_VEL
LIN {X 0,Y 325.121,Z 200.896,A -85,B 0,C 180,E1 -15322.898,E2 -15322.898} C_VEL
LIN {X 0,Y 328.207,Z 213.252,A -85,B 0,C 180,E1 -15324.158,E2 -15324.158} C_VEL
LIN {X 0,Y 328.58,Z 216.78,A -85,B 0,C 180,E1 -15324.523,E2 -15324.523} C_VEL
LIN {X 0,Y 327.218,Z 228.559,A -85,B 0,C 180,E1 -15325.718,E2 -15325.718} C_VEL
LIN {X 0,Y 325.93,Z 238.049,A -85,B 0,C 180,E1 -15326.924,E2 -15326.924} C_VEL
LIN {X 0,Y 324.463,Z 247.808,A -85,B 0,C 180,E1 -15328.458,E2 -15328.458} C_VEL
LIN {X 0,Y 323.165,Z 255.86,A -85,B 0,C 180,E1 -15330.012,E2 -15330.012} C_VEL
LIN {X 0,Y 321.736,Z 264.131,A -85,B 0,C 180,E1 -15331.985,E2 -15331.985} C_VEL
LIN {X 0,Y 320.701,Z 269.616,A -85,B 0,C 180,E1 -15333.617,E2 -15333.617} C_VEL
LIN {X 0,Y 319.836,Z 274.961,A -85,B 0,C 180,E1 -15335.606,E2 -15335.606} C_VEL
LIN {X 0,Y 319.131,Z 278.945,A -85,B 0,C 180,E1 -15337.551,E2 -15337.551} C_VEL
LIN {X 0,Y 318.485,Z 282.155,A -85,B 0,C 180,E1 -15339.787,E2 -15339.787} C_VEL
LIN {X 0,Y 318.179,Z 283.744,A -85,B 0,C 180,E1 -15341.501,E2 -15341.501} C_VEL
LIN {X 0,Y 317.944,Z 284.56,A -85,B 0,C 180,E1 -15343.253,E2 -15343.253} C_VEL
LIN {X 0,Y 317.886,Z 284.607,A -85,B 0,C 180,E1 -15345.029,E2 -15345.029} C_VEL
LIN {X 0,Y 317.89,Z 283.85,A -85,B 0,C 180,E1 -15346.849,E2 -15346.849} C_VEL
LIN {X 0,Y 318.099,Z 282.229,A -85,B 0,C 180,E1 -15348.692,E2 -15348.692} C_VEL
LIN {X 0,Y 318.448,Z 279.652,A -85,B 0,C 180,E1 -15350.572,E2 -15350.572} C_VEL
LIN {X 0,Y 318.856,Z 275.945,A -85,B 0,C 180,E1 -15352.511,E2 -15352.511} C_VEL
LIN {X 0,Y 319.492,Z 270.973,A -85,B 0,C 180,E1 -15354.478,E2 -15354.478} C_VEL
LIN {X 0,Y 320.251,Z 264.432,A -85,B 0,C 180,E1 -15356.502,E2 -15356.502} C_VEL
LIN {X 0,Y 321.366,Z 256.145,A -85,B 0,C 180,E1 -15358.527,E2 -15358.527} C_VEL
LIN {X 0,Y 322.553,Z 246.99,A -85,B 0,C 180,E1 -15360.297,E2 -15360.297} C_VEL
LIN {X 0,Y 323.718,Z 236.519,A -85,B 0,C 180,E1 -15361.937,E2 -15361.937} C_VEL
LIN {X 0,Y 324.923,Z 225.226,A -85,B 0,C 180,E1 -15363.332,E2 -15363.332} C_VEL
LIN {X 0,Y 326.048,Z 213.647,A -85,B 0,C 180,E1 -15364.462,E2 -15364.462} C_VEL
LIN {X 0,Y 325.857,Z 210.038,A -85,B 0,C 180,E1 -15364.788,E2 -15364.788} C_VEL
LIN {X 0,Y 323.41,Z 198.525,A -85,B 0,C 180,E1 -15365.784,E2 -15365.784} C_VEL
LIN {X 0,Y 320.073,Z 185.88,A -85,B 0,C 180,E1 -15366.676,E2 -15366.676} C_VEL
LIN {X 0,Y 318.598,Z 180.522,A -85,B 0,C 180,E1 -15366.992,E2 -15366.992} C_VEL
LIN {X 0,Y 318.729,Z 177.14,A -85,B 0,C 180,E1 -15370.685,E2 -15370.685} C_VEL
LIN {X 0,Y 318.931,Z 173.597,A -85,B 0,C 180,E1 -15374.666,E2 -15374.666} C_VEL
LIN {X 0,Y 319.089,Z 172.74,A -85,B 0,C 180,E1 -15375.979,E2 -15375.979} C_VEL
LIN {X 0,Y 319.563,Z 172.678,A -85,B 0,C 180,E1 -15379.866,E2 -15379.866} C_VEL
LIN {X 0,Y 319.888,Z 172.639,A -85,B 0,C 180,E1 -15382.425,E2 -15382.425} C_VEL
LIN {X 0,Y 319.739,Z 172.654,A -85,B 0,C 180,E1 -15384.956,E2 -15384.956} C_VEL
LIN {X 0,Y 319.988,Z 172.624,A -85,B 0,C 180,E1 -15387.482,E2 -15387.482} C_VEL
LIN {X 0,Y 320.165,Z 172.606,A -85,B 0,C 180,E1 -15390,E2 -15390} C_VEL
LIN {X 0,Y 319.988,Z 172.624,A -85,B 0,C 180,E1 -15392.517,E2 -15392.517} C_VEL
LIN {X 0,Y 319.948,Z 172.63,A -85,B 0,C 180,E1 -15396.305,E2 -15396.305} C_VEL
LIN {X 0,Y 319.839,Z 172.642,A -85,B 0,C 180,E1 -15398.848,E2 -15398.848} C_VEL
LIN {X 0,Y 319.678,Z 172.662,A -85,B 0,C 180,E1 -15402.7,E2 -15402.7} C_VEL
LIN {X 0,Y 319.696,Z 172.662,A -85,B 0,C 180,E1 -15405.296,E2 -15405.296} C_VEL
LIN {X 0,Y 319.67,Z 172.665,A -85,B 0,C 180,E1 -15409.255,E2 -15409.255} C_VEL
LIN {X 0,Y 319.567,Z 172.679,A -85,B 0,C 180,E1 -15413.32,E2 -15413.32} C_VEL
LIN {X 0,Y 319.615,Z 172.67,A -85,B 0,C 180,E1 -15416.09,E2 -15416.09} C_VEL
LIN {X 0,Y 319.576,Z 172.676,A -85,B 0,C 180,E1 -15418.935,E2 -15418.935} C_VEL
LIN {X 0,Y 319.527,Z 172.682,A -85,B 0,C 180,E1 -15421.862,E2 -15421.862} C_VEL
LIN {X 0,Y 319.577,Z 172.676,A -85,B 0,C 180,E1 -15425.543,E2 -15425.543} C_VEL
LIN {X 0,Y 319.555,Z 172.678,A -85,B 0,C 180,E1 -15429.669,E2 -15429.669} C_VEL
LIN {X 0,Y 319.554,Z 172.679,A -85,B 0,C 180,E1 -15433.468,E2 -15433.468} C_VEL
LIN {X 0,Y 319.558,Z 172.681,A -85,B 0,C 180,E1 -15437.018,E2 -15437.018} C_VEL
LIN {X 0,Y 319.544,Z 172.679,A -85,B 0,C 180,E1 -15440.371,E2 -15440.371} C_VEL
LIN {X 0,Y 319.578,Z 172.676,A -85,B 0,C 180,E1 -15444.457,E2 -15444.457} C_VEL
LIN {X 0,Y 319.529,Z 172.681,A -85,B 0,C 180,E1 -15448.139,E2 -15448.139} C_VEL
LIN {X 0,Y 319.609,Z 172.669,A -85,B 0,C 180,E1 -15451.591,E2 -15451.591} C_VEL
LIN {X 0,Y 319.604,Z 172.671,A -85,B 0,C 180,E1 -15455.305,E2 -15455.305} C_VEL
LIN {X 0,Y 319.568,Z 172.679,A -85,B 0,C 180,E1 -15456.629,E2 -15456.629} C_VEL
LIN {X 0,Y 318.945,Z 172.764,A -85,B 0,C 180,E1 -15457.682,E2 -15457.682} C_VEL
LIN {X 0,Y 316.145,Z 173.112,A -85,B 0,C 180,E1 -15459.396,E2 -15459.396} C_VEL
LIN {X 0,Y 313.741,Z 173.404,A -85,B 0,C 180,E1 -15460.786,E2 -15460.786} C_VEL
LIN {X 0,Y 312.695,Z 173.532,A -85,B 0,C 180,E1 -15461.861,E2 -15461.861} C_VEL
LIN {X 0,Y 312.604,Z 173.54,A -85,B 0,C 180,E1 -15462.225,E2 -15462.225} C_VEL
LIN {X 0,Y 312.694,Z 173.531,A -85,B 0,C 180,E1 -15465.687,E2 -15465.687} C_VEL
LIN {X 0,Y 312.699,Z 173.532,A -85,B 0,C 180,E1 -15469.642,E2 -15469.642} C_VEL
LIN {X 0,Y 312.853,Z 173.517,A -85,B 0,C 180,E1 -15472.254,E2 -15472.254} C_VEL
LIN {X 0,Y 312.716,Z 173.529,A -85,B 0,C 180,E1 -15474.843,E2 -15474.843} C_VEL
LIN {X 0,Y 312.99,Z 173.495,A -85,B 0,C 180,E1 -15478.714,E2 -15478.714} C_VEL
LIN {X 0,Y 312.99,Z 173.495,A -85,B 0,C 180,E1 -15481.287,E2 -15481.287} C_VEL
LIN {X 0,Y 312.707,Z 173.53,A -85,B 0,C 180,E1 -15485.158,E2 -15485.158} C_VEL
LIN {X 0,Y 312.819,Z 173.52,A -85,B 0,C 180,E1 -15487.748,E2 -15487.748} C_VEL
LIN {X 0,Y 312.665,Z 173.539,A -85,B 0,C 180,E1 -15491.672,E2 -15491.672} C_VEL
LIN {X 0,Y 312.702,Z 173.531,A -85,B 0,C 180,E1 -15494.888,E2 -15494.888} C_VEL
LIN {X 0,Y 312.632,Z 173.541,A -85,B 0,C 180,E1 -15499.237,E2 -15499.237} C_VEL
LIN {X 0,Y 312.548,Z 173.55,A -85,B 0,C 180,E1 -15502.79,E2 -15502.79} C_VEL
LIN {X 0,Y 312.599,Z 173.545,A -85,B 0,C 180,E1 -15505.934,E2 -15505.934} C_VEL
LIN {X 0,Y 312.54,Z 173.554,A -85,B 0,C 180,E1 -15509.651,E2 -15509.651} C_VEL
LIN {X 0,Y 312.521,Z 173.556,A -85,B 0,C 180,E1 -15513.689,E2 -15513.689} C_VEL
LIN {X 0,Y 312.527,Z 173.557,A -85,B 0,C 180,E1 -15517.386,E2 -15517.386} C_VEL
LIN {X 0,Y 312.534,Z 173.652,A -85,B 0,C 180,E1 -15521.129,E2 -15521.129} C_VEL
LIN {X 0,Y 313.468,Z 178.712,A -85,B 0,C 180,E1 -15524.929,E2 -15524.929} C_VEL
LIN {X 0,Y 314.456,Z 184.034,A -85,B 0,C 180,E1 -15528.706,E2 -15528.706} C_VEL
LIN {X 0,Y 315.111,Z 187.989,A -85,B 0,C 180,E1 -15531.355,E2 -15531.355} C_VEL
LIN {X 0,Y 315.314,Z 191.137,A -85,B 0,C 180,E1 -15533.361,E2 -15533.361} C_VEL
LIN {X 0,Y 314.588,Z 196.862,A -85,B 0,C 180,E1 -15536.816,E2 -15536.816} C_VEL
LIN {X 0,Y 313.55,Z 203.994,A -85,B 0,C 180,E1 -15540.946,E2 -15540.946} C_VEL
LIN {X 0,Y 312.733,Z 210.657,A -85,B 0,C 180,E1 -15544.724,E2 -15544.724} C_VEL
LIN {X 0,Y 312.251,Z 215.057,A -85,B 0,C 180,E1 -15547.17,E2 -15547.17} C_VEL
LIN {X 0,Y 314.65,Z 228.902,A -85,B 0,C 180,E1 -15547.918,E2 -15547.918} C_VEL
LIN {X 0,Y 316.447,Z 241.966,A -85,B 0,C 180,E1 -15548.874,E2 -15548.874} C_VEL
LIN {X 0,Y 317.55,Z 253.607,A -85,B 0,C 180,E1 -15549.938,E2 -15549.938} C_VEL
LIN {X 0,Y 317.943,Z 260.178,A -85,B 0,C 180,E1 -15550.636,E2 -15550.636} C_VEL
LIN {X 0,Y 316.489,Z 270.784,A -85,B 0,C 180,E1 -15551.888,E2 -15551.888} C_VEL
LIN {X 0,Y 315.211,Z 280.752,A -85,B 0,C 180,E1 -15553.357,E2 -15553.357} C_VEL
LIN {X 0,Y 313.994,Z 290.241,A -85,B 0,C 180,E1 -15555.084,E2 -15555.084} C_VEL
LIN {X 0,Y 312.795,Z 298.737,A -85,B 0,C 180,E1 -15557.016,E2 -15557.016} C_VEL
LIN {X 0,Y 311.945,Z 305.567,A -85,B 0,C 180,E1 -15558.96,E2 -15558.96} C_VEL
LIN {X 0,Y 311.376,Z 311.028,A -85,B 0,C 180,E1 -15560.91,E2 -15560.91} C_VEL
LIN {X 0,Y 311.006,Z 315.285,A -85,B 0,C 180,E1 -15562.861,E2 -15562.861} C_VEL
LIN {X 0,Y 310.865,Z 318.46,A -85,B 0,C 180,E1 -15564.812,E2 -15564.812} C_VEL
LIN {X 0,Y 310.844,Z 320.03,A -85,B 0,C 180,E1 -15566.111,E2 -15566.111} C_VEL
LIN {X 0,Y 310.785,Z 321.163,A -85,B 0,C 180,E1 -15567.408,E2 -15567.408} C_VEL
LIN {X 0,Y 310.852,Z 321.859,A -85,B 0,C 180,E1 -15568.705,E2 -15568.705} C_VEL
LIN {X 0,Y 310.954,Z 322.159,A -85,B 0,C 180,E1 -15570,E2 -15570} C_VEL
LIN {X 0,Y 310.842,Z 322.049,A -85,B 0,C 180,E1 -15571.296,E2 -15571.296} C_VEL
LIN {X 0,Y 310.775,Z 321.533,A -85,B 0,C 180,E1 -15572.593,E2 -15572.593} C_VEL
LIN {X 0,Y 310.814,Z 320.582,A -85,B 0,C 180,E1 -15573.89,E2 -15573.89} C_VEL
LIN {X 0,Y 310.89,Z 318.299,A -85,B 0,C 180,E1 -15575.914,E2 -15575.914} C_VEL
LIN {X 0,Y 311.203,Z 313.964,A -85,B 0,C 180,E1 -15578.441,E2 -15578.441} C_VEL
LIN {X 0,Y 311.725,Z 309.388,A -85,B 0,C 180,E1 -15580.391,E2 -15580.391} C_VEL
LIN {X 0,Y 312.667,Z 302.523,A -85,B 0,C 180,E1 -15582.66,E2 -15582.66} C_VEL
LIN {X 0,Y 313.924,Z 295.12,A -85,B 0,C 180,E1 -15584.588,E2 -15584.588} C_VEL
LIN {X 0,Y 315.228,Z 286.852,A -85,B 0,C 180,E1 -15586.342,E2 -15586.342} C_VEL
LIN {X 0,Y 316.732,Z 276.641,A -85,B 0,C 180,E1 -15588.099,E2 -15588.099} C_VEL
LIN {X 0,Y 318.603,Z 265.072,A -85,B 0,C 180,E1 -15589.658,E2 -15589.658} C_VEL
LIN {X 0,Y 319.077,Z 259.621,A -85,B 0,C 180,E1 -15590.299,E2 -15590.299} C_VEL
LIN {X 0,Y 318.529,Z 247.236,A -85,B 0,C 180,E1 -15591.628,E2 -15591.628} C_VEL
LIN {X 0,Y 317.195,Z 234.111,A -85,B 0,C 180,E1 -15592.794,E2 -15592.794} C_VEL
LIN {X 0,Y 314.698,Z 221.712,A -85,B 0,C 180,E1 -15593.762,E2 -15593.762} C_VEL
LIN {X 0,Y 312.54,Z 212.899,A -85,B 0,C 180,E1 -15594.352,E2 -15594.352} C_VEL
LIN {X 0,Y 313.365,Z 206.41,A -85,B 0,C 180,E1 -15598.098,E2 -15598.098} C_VEL
LIN {X 0,Y 314.356,Z 200.201,A -85,B 0,C 180,E1 -15601.835,E2 -15601.835} C_VEL
LIN {X 0,Y 315.338,Z 194.575,A -85,B 0,C 180,E1 -15605.413,E2 -15605.413} C_VEL
LIN {X 0,Y 315.544,Z 191.137,A -85,B 0,C 180,E1 -15607.771,E2 -15607.771} C_VEL
LIN {X 0,Y 315.021,Z 187.313,A -85,B 0,C 180,E1 -15610.665,E2 -15610.665} C_VEL
LIN {X 0,Y 314.206,Z 182.968,A -85,B 0,C 180,E1 -15614.294,E2 -15614.294} C_VEL
LIN {X 0,Y 313.556,Z 179.319,A -85,B 0,C 180,E1 -15617.745,E2 -15617.745} C_VEL
LIN {X 0,Y 312.917,Z 175.638,A -85,B 0,C 180,E1 -15621.822,E2 -15621.822} C_VEL
LIN {X 0,Y 312.535,Z 173.556,A -85,B 0,C 180,E1 -15624.616,E2 -15624.616} C_VEL
LIN {X 0,Y 312.524,Z 173.555,A -85,B 0,C 180,E1 -15628.853,E2 -15628.853} C_VEL
LIN {X 0,Y 312.574,Z 173.55,A -85,B 0,C 180,E1 -15631.824,E2 -15631.824} C_VEL
LIN {X 0,Y 312.59,Z 173.547,A -85,B 0,C 180,E1 -15634.711,E2 -15634.711} C_VEL
LIN {X 0,Y 312.591,Z 173.545,A -85,B 0,C 180,E1 -15637.529,E2 -15637.529} C_VEL
LIN {X 0,Y 312.593,Z 173.544,A -85,B 0,C 180,E1 -15641.653,E2 -15641.653} C_VEL
LIN {X 0,Y 312.689,Z 173.536,A -85,B 0,C 180,E1 -15645.685,E2 -15645.685} C_VEL
LIN {X 0,Y 312.706,Z 173.534,A -85,B 0,C 180,E1 -15649.641,E2 -15649.641} C_VEL
LIN {X 0,Y 312.876,Z 173.513,A -85,B 0,C 180,E1 -15652.254,E2 -15652.254} C_VEL
LIN {X 0,Y 312.722,Z 173.533,A -85,B 0,C 180,E1 -15654.842,E2 -15654.842} C_VEL
LIN {X 0,Y 312.995,Z 173.499,A -85,B 0,C 180,E1 -15658.713,E2 -15658.713} C_VEL
LIN {X 0,Y 313.124,Z 173.483,A -85,B 0,C 180,E1 -15659.999,E2 -15659.999} C_VEL
LIN {X 0,Y 312.941,Z 173.504,A -85,B 0,C 180,E1 -15662.574,E2 -15662.574} C_VEL
LIN {X 0,Y 312.728,Z 173.666,A -85,B 0,C 180,E1 -15665.157,E2 -15665.157} C_VEL
LIN {X 0,Y 313.076,Z 175.102,A -85,B 0,C 180,E1 -15667.74,E2 -15667.74} C_VEL
LIN {X 0,Y 312.854,Z 177.613,A -85,B 0,C 180,E1 -15671.664,E2 -15671.664} C_VEL
LIN {X 0,Y 312.614,Z 179.779,A -85,B 0,C 180,E1 -15674.826,E2 -15674.826} C_VEL
LIN {X 0,Y 312.249,Z 182.831,A -85,B 0,C 180,E1 -15679.034,E2 -15679.034} C_VEL
LIN {X 0,Y 312.125,Z 184.077,A -85,B 0,C 180,E1 -15680.684,E2 -15680.684} C_VEL
LIN {X 0,Y 314.221,Z 189.712,A -85,B 0,C 180,E1 -15681.183,E2 -15681.183} C_VEL
LIN {X 0,Y 318.279,Z 201.37,A -85,B 0,C 180,E1 -15682.296,E2 -15682.296} C_VEL
LIN {X 0,Y 320.962,Z 211.785,A -85,B 0,C 180,E1 -15683.382,E2 -15683.382} C_VEL
LIN {X 0,Y 322.066,Z 217.004,A -85,B 0,C 180,E1 -15683.98,E2 -15683.98} C_VEL
LIN {X 0,Y 320.821,Z 227.991,A -85,B 0,C 180,E1 -15685.114,E2 -15685.114} C_VEL
LIN {X 0,Y 319.321,Z 238.537,A -85,B 0,C 180,E1 -15686.466,E2 -15686.466} C_VEL
LIN {X 0,Y 317.732,Z 248.662,A -85,B 0,C 180,E1 -15688.1,E2 -15688.1} C_VEL
LIN {X 0,Y 316.189,Z 257.65,A -85,B 0,C 180,E1 -15689.903,E2 -15689.903} C_VEL
LIN {X 0,Y 314.895,Z 264.701,A -85,B 0,C 180,E1 -15691.654,E2 -15691.654} C_VEL
LIN {X 0,Y 313.666,Z 270.932,A -85,B 0,C 180,E1 -15693.58,E2 -15693.58} C_VEL
LIN {X 0,Y 312.715,Z 276.343,A -85,B 0,C 180,E1 -15695.755,E2 -15695.755} C_VEL
LIN {X 0,Y 311.916,Z 280.394,A -85,B 0,C 180,E1 -15697.944,E2 -15697.944} C_VEL
LIN {X 0,Y 311.38,Z 282.892,A -85,B 0,C 180,E1 -15699.879,E2 -15699.879} C_VEL
LIN {X 0,Y 311.054,Z 284.432,A -85,B 0,C 180,E1 -15701.788,E2 -15701.788} C_VEL
LIN {X 0,Y 310.797,Z 285.128,A -85,B 0,C 180,E1 -15704.506,E2 -15704.506} C_VEL
LIN {X 0,Y 310.785,Z 284.568,A -85,B 0,C 180,E1 -15706.355,E2 -15706.355} C_VEL
LIN {X 0,Y 310.944,Z 283.146,A -85,B 0,C 180,E1 -15708.233,E2 -15708.233} C_VEL
LIN {X 0,Y 311.405,Z 279.776,A -85,B 0,C 180,E1 -15710.807,E2 -15710.807} C_VEL
LIN {X 0,Y 311.779,Z 276.593,A -85,B 0,C 180,E1 -15712.509,E2 -15712.509} C_VEL
LIN {X 0,Y 312.47,Z 271.43,A -85,B 0,C 180,E1 -15714.608,E2 -15714.608} C_VEL
LIN {X 0,Y 313.308,Z 264.392,A -85,B 0,C 180,E1 -15716.819,E2 -15716.819} C_VEL
LIN {X 0,Y 314.336,Z 256.988,A -85,B 0,C 180,E1 -15718.663,E2 -15718.663} C_VEL
LIN {X 0,Y 315.456,Z 248.75,A -85,B 0,C 180,E1 -15720.327,E2 -15720.327} C_VEL
LIN {X 0,Y 316.722,Z 238.231,A -85,B 0,C 180,E1 -15722.046,E2 -15722.046} C_VEL
LIN {X 0,Y 317.92,Z 227.878,A -85,B 0,C 180,E1 -15723.407,E2 -15723.407} C_VEL
LIN {X 0,Y 319,Z 216.577,A -85,B 0,C 180,E1 -15724.591,E2 -15724.591} C_VEL
LIN {X 0,Y 319.27,Z 212.644,A -85,B 0,C 180,E1 -15724.95,E2 -15724.95} C_VEL
LIN {X 0,Y 316.641,Z 199.942,A -85,B 0,C 180,E1 -15726.104,E2 -15726.104} C_VEL
LIN {X 0,Y 313.232,Z 186.952,A -85,B 0,C 180,E1 -15727.066,E2 -15727.066} C_VEL
LIN {X 0,Y 311.559,Z 180.901,A -85,B 0,C 180,E1 -15727.45,E2 -15727.45} C_VEL
LIN {X 0,Y 311.721,Z 177.167,A -85,B 0,C 180,E1 -15731.6,E2 -15731.6} C_VEL
LIN {X 0,Y 311.976,Z 173.626,A -85,B 0,C 180,E1 -15735.652,E2 -15735.652} C_VEL
LIN {X 0,Y 312.477,Z 173.559,A -85,B 0,C 180,E1 -15739.634,E2 -15739.634} C_VEL
LIN {X 0,Y 312.824,Z 173.521,A -85,B 0,C 180,E1 -15742.253,E2 -15742.253} C_VEL
LIN {X 0,Y 312.887,Z 173.509,A -85,B 0,C 180,E1 -15743.551,E2 -15743.551} C_VEL
LIN {X 0,Y 312.934,Z 173.502,A -85,B 0,C 180,E1 -15747.425,E2 -15747.425} C_VEL
LIN {X 0,Y 313.117,Z 173.484,A -85,B 0,C 180,E1 -15750,E2 -15750} C_VEL
LIN {X 0,Y 312.935,Z 173.502,A -85,B 0,C 180,E1 -15752.574,E2 -15752.574} C_VEL
LIN {X 0,Y 312.906,Z 173.506,A -85,B 0,C 180,E1 -15756.448,E2 -15756.448} C_VEL
LIN {X 0,Y 312.784,Z 173.521,A -85,B 0,C 180,E1 -15759.049,E2 -15759.049} C_VEL
LIN {X 0,Y 312.631,Z 173.54,A -85,B 0,C 180,E1 -15762.991,E2 -15762.991} C_VEL
LIN {X 0,Y 312.635,Z 173.545,A -85,B 0,C 180,E1 -15765.65,E2 -15765.65} C_VEL
LIN {X 0,Y 312.626,Z 173.542,A -85,B 0,C 180,E1 -15769.236,E2 -15769.236} C_VEL
LIN {X 0,Y 312.542,Z 173.551,A -85,B 0,C 180,E1 -15772.789,E2 -15772.789} C_VEL
LIN {X 0,Y 312.593,Z 173.545,A -85,B 0,C 180,E1 -15775.934,E2 -15775.934} C_VEL
LIN {X 0,Y 312.535,Z 173.555,A -85,B 0,C 180,E1 -15779.651,E2 -15779.651} C_VEL
LIN {X 0,Y 312.516,Z 173.555,A -85,B 0,C 180,E1 -15783.689,E2 -15783.689} C_VEL
LIN {X 0,Y 312.517,Z 173.557,A -85,B 0,C 180,E1 -15787.386,E2 -15787.386} C_VEL
LIN {X 0,Y 312.487,Z 173.559,A -85,B 0,C 180,E1 -15790.709,E2 -15790.709} C_VEL
LIN {X 0,Y 312.47,Z 173.559,A -85,B 0,C 180,E1 -15794.206,E2 -15794.206} C_VEL
LIN {X 0,Y 312.483,Z 173.556,A -85,B 0,C 180,E1 -15797.919,E2 -15797.919} C_VEL
LIN {X 0,Y 312.496,Z 173.561,A -85,B 0,C 180,E1 -15800.972,E2 -15800.972} C_VEL
LIN {X 0,Y 312.53,Z 173.553,A -85,B 0,C 180,E1 -15804.221,E2 -15804.221} C_VEL
LIN {X 0,Y 312.502,Z 173.556,A -85,B 0,C 180,E1 -15807.334,E2 -15807.334} C_VEL
LIN {X 0,Y 312.543,Z 173.55,A -85,B 0,C 180,E1 -15811.279,E2 -15811.279} C_VEL
LIN {X 0,Y 312.584,Z 173.549,A -85,B 0,C 180,E1 -15814.712,E2 -15814.712} C_VEL
LIN {X 0,Y 312.587,Z 173.545,A -85,B 0,C 180,E1 -15817.53,E2 -15817.53} C_VEL
LIN {X 0,Y 312.638,Z 173.538,A -85,B 0,C 180,E1 -15821.657,E2 -15821.657} C_VEL
LIN {X 0,Y 312.604,Z 173.54,A -85,B 0,C 180,E1 -15822.225,E2 -15822.225} C_VEL
LIN {X 0,Y 311.912,Z 173.628,A -85,B 0,C 180,E1 -15823.301,E2 -15823.301} C_VEL
LIN {X 0,Y 309.038,Z 173.986,A -85,B 0,C 180,E1 -15825.052,E2 -15825.052} C_VEL
LIN {X 0,Y 306.643,Z 174.289,A -85,B 0,C 180,E1 -15826.472,E2 -15826.472} C_VEL
LIN {X 0,Y 305.655,Z 174.408,A -85,B 0,C 180,E1 -15827.571,E2 -15827.571} C_VEL
LIN {X 0,Y 305.596,Z 174.417,A -85,B 0,C 180,E1 -15827.943,E2 -15827.943} C_VEL
LIN {X 0,Y 305.797,Z 174.395,A -85,B 0,C 180,E1 -15832.075,E2 -15832.075} C_VEL
LIN {X 0,Y 305.687,Z 174.404,A -85,B 0,C 180,E1 -15834.724,E2 -15834.724} C_VEL
LIN {X 0,Y 305.957,Z 174.37,A -85,B 0,C 180,E1 -15838.684,E2 -15838.684} C_VEL
LIN {X 0,Y 305.957,Z 174.371,A -85,B 0,C 180,E1 -15841.317,E2 -15841.317} C_VEL
LIN {X 0,Y 305.676,Z 174.406,A -85,B 0,C 180,E1 -15845.277,E2 -15845.277} C_VEL
LIN {X 0,Y 305.765,Z 174.398,A -85,B 0,C 180,E1 -15847.928,E2 -15847.928} C_VEL
LIN {X 0,Y 305.601,Z 174.419,A -85,B 0,C 180,E1 -15851.946,E2 -15851.946} C_VEL
LIN {X 0,Y 305.639,Z 174.411,A -85,B 0,C 180,E1 -15855.036,E2 -15855.036} C_VEL
LIN {X 0,Y 305.579,Z 174.421,A -85,B 0,C 180,E1 -15859.446,E2 -15859.446} C_VEL
LIN {X 0,Y 305.493,Z 174.43,A -85,B 0,C 180,E1 -15863.042,E2 -15863.042} C_VEL
LIN {X 0,Y 305.528,Z 174.425,A -85,B 0,C 180,E1 -15866.219,E2 -15866.219} C_VEL
LIN {X 0,Y 305.49,Z 174.432,A -85,B 0,C 180,E1 -15869.048,E2 -15869.048} C_VEL
LIN {X 0,Y 305.444,Z 174.436,A -85,B 0,C 180,E1 -15871.953,E2 -15871.953} C_VEL
LIN {X 0,Y 305.464,Z 174.437,A -85,B 0,C 180,E1 -15875.114,E2 -15875.114} C_VEL
LIN {X 0,Y 305.451,Z 174.437,A -85,B 0,C 180,E1 -15878.529,E2 -15878.529} C_VEL
LIN {X 0,Y 305.495,Z 174.508,A -85,B 0,C 180,E1 -15880.7,E2 -15880.7} C_VEL
LIN {X 0,Y 306.44,Z 179.667,A -85,B 0,C 180,E1 -15884.687,E2 -15884.687} C_VEL
LIN {X 0,Y 307.539,Z 185.559,A -85,B 0,C 180,E1 -15888.95,E2 -15888.95} C_VEL
LIN {X 0,Y 308.227,Z 190.074,A -85,B 0,C 180,E1 -15892.002,E2 -15892.002} C_VEL
LIN {X 0,Y 308.089,Z 193.871,A -85,B 0,C 180,E1 -15894.43,E2 -15894.43} C_VEL
LIN {X 0,Y 307.272,Z 199.425,A -85,B 0,C 180,E1 -15897.81,E2 -15897.81} C_VEL
LIN {X 0,Y 306.236,Z 206.4,A -85,B 0,C 180,E1 -15901.936,E2 -15901.936} C_VEL
LIN {X 0,Y 305.336,Z 213.905,A -85,B 0,C 180,E1 -15906.247,E2 -15906.247} C_VEL
LIN {X 0,Y 305.254,Z 214.688,A -85,B 0,C 180,E1 -15906.694,E2 -15906.694} C_VEL
LIN {X 0,Y 307.791,Z 229.31,A -85,B 0,C 180,E1 -15907.525,E2 -15907.525} C_VEL
LIN {X 0,Y 309.594,Z 242.746,A -85,B 0,C 180,E1 -15908.55,E2 -15908.55} C_VEL
LIN {X 0,Y 310.671,Z 254.565,A -85,B 0,C 180,E1 -15909.681,E2 -15909.681} C_VEL
LIN {X 0,Y 310.995,Z 260.605,A -85,B 0,C 180,E1 -15910.358,E2 -15910.358} C_VEL
LIN {X 0,Y 309.343,Z 272.214,A -85,B 0,C 180,E1 -15911.797,E2 -15911.797} C_VEL
LIN {X 0,Y 308.097,Z 282.155,A -85,B 0,C 180,E1 -15913.35,E2 -15913.35} C_VEL
LIN {X 0,Y 306.843,Z 291.051,A -85,B 0,C 180,E1 -15915.068,E2 -15915.068} C_VEL
LIN {X 0,Y 305.669,Z 299.301,A -85,B 0,C 180,E1 -15917.046,E2 -15917.046} C_VEL
LIN {X 0,Y 304.818,Z 305.953,A -85,B 0,C 180,E1 -15919.035,E2 -15919.035} C_VEL
LIN {X 0,Y 304.163,Z 312.012,A -85,B 0,C 180,E1 -15921.362,E2 -15921.362} C_VEL
LIN {X 0,Y 303.855,Z 315.935,A -85,B 0,C 180,E1 -15923.359,E2 -15923.359} C_VEL
LIN {X 0,Y 303.784,Z 317.947,A -85,B 0,C 180,E1 -15924.69,E2 -15924.69} C_VEL
LIN {X 0,Y 303.777,Z 319.536,A -85,B 0,C 180,E1 -15926.02,E2 -15926.02} C_VEL
LIN {X 0,Y 303.707,Z 320.697,A -85,B 0,C 180,E1 -15927.348,E2 -15927.348} C_VEL
LIN {X 0,Y 303.76,Z 321.411,A -85,B 0,C 180,E1 -15928.674,E2 -15928.674} C_VEL
LIN {X 0,Y 303.866,Z 321.726,A -85,B 0,C 180,E1 -15930,E2 -15930} C_VEL
LIN {X 0,Y 303.749,Z 321.63,A -85,B 0,C 180,E1 -15931.326,E2 -15931.326} C_VEL
LIN {X 0,Y 303.697,Z 321.139,A -85,B 0,C 180,E1 -15932.653,E2 -15932.653} C_VEL
LIN {X 0,Y 303.724,Z 320.207,A -85,B 0,C 180,E1 -15933.981,E2 -15933.981} C_VEL
LIN {X 0,Y 303.812,Z 318.176,A -85,B 0,C 180,E1 -15935.892,E2 -15935.892} C_VEL
LIN {X 0,Y 304.018,Z 314.942,A -85,B 0,C 180,E1 -15937.973,E2 -15937.973} C_VEL
LIN {X 0,Y 304.483,Z 310.782,A -85,B 0,C 180,E1 -15939.969,E2 -15939.969} C_VEL
LIN {X 0,Y 305.383,Z 304.453,A -85,B 0,C 180,E1 -15942.291,E2 -15942.291} C_VEL
LIN {X 0,Y 306.57,Z 297.62,A -85,B 0,C 180,E1 -15944.267,E2 -15944.267} C_VEL
LIN {X 0,Y 308.027,Z 289.125,A -85,B 0,C 180,E1 -15946.247,E2 -15946.247} C_VEL
LIN {X 0,Y 309.355,Z 280.611,A -85,B 0,C 180,E1 -15947.861,E2 -15947.861} C_VEL
LIN {X 0,Y 311.133,Z 270.119,A -85,B 0,C 180,E1 -15949.462,E2 -15949.462} C_VEL
LIN {X 0,Y 312.344,Z 261.245,A -85,B 0,C 180,E1 -15950.584,E2 -15950.584} C_VEL
LIN {X 0,Y 312.011,Z 249.823,A -85,B 0,C 180,E1 -15951.903,E2 -15951.903} C_VEL
LIN {X 0,Y 311.104,Z 238.371,A -85,B 0,C 180,E1 -15953.018,E2 -15953.018} C_VEL
LIN {X 0,Y 308.931,Z 225.857,A -85,B 0,C 180,E1 -15954.087,E2 -15954.087} C_VEL
LIN {X 0,Y 305.623,Z 212.351,A -85,B 0,C 180,E1 -15955.103,E2 -15955.103} C_VEL
LIN {X 0,Y 306.491,Z 206.193,A -85,B 0,C 180,E1 -15958.787,E2 -15958.787} C_VEL
LIN {X 0,Y 307.412,Z 200.659,A -85,B 0,C 180,E1 -15962.232,E2 -15962.232} C_VEL
LIN {X 0,Y 308.342,Z 195.609,A -85,B 0,C 180,E1 -15965.536,E2 -15965.536} C_VEL
LIN {X 0,Y 308.562,Z 192.191,A -85,B 0,C 180,E1 -15967.95,E2 -15967.95} C_VEL
LIN {X 0,Y 307.875,Z 187.734,A -85,B 0,C 180,E1 -15971.453,E2 -15971.453} C_VEL
LIN {X 0,Y 307.091,Z 183.538,A -85,B 0,C 180,E1 -15975.191,E2 -15975.191} C_VEL
LIN {X 0,Y 306.508,Z 180.386,A -85,B 0,C 180,E1 -15978.321,E2 -15978.321} C_VEL
LIN {X 0,Y 306.032,Z 177.434,A -85,B 0,C 180,E1 -15981.679,E2 -15981.679} C_VEL
LIN {X 0,Y 305.493,Z 174.585,A -85,B 0,C 180,E1 -15985.467,E2 -15985.467} C_VEL
LIN {X 0,Y 305.462,Z 174.434,A -85,B 0,C 180,E1 -15989.59,E2 -15989.59} C_VEL
LIN {X 0,Y 305.523,Z 174.427,A -85,B 0,C 180,E1 -15992.608,E2 -15992.608} C_VEL
LIN {X 0,Y 305.512,Z 174.427,A -85,B 0,C 180,E1 -15995.538,E2 -15995.538} C_VEL
LIN {X 0,Y 305.516,Z 174.426,A -85,B 0,C 180,E1 -15999.814,E2 -15999.814} C_VEL
LIN {X 0,Y 305.548,Z 174.423,A -85,B 0,C 180,E1 -16002.601,E2 -16002.601} C_VEL
LIN {X 0,Y 305.63,Z 174.415,A -85,B 0,C 180,E1 -16005.347,E2 -16005.347} C_VEL
LIN {X 0,Y 305.643,Z 174.414,A -85,B 0,C 180,E1 -16009.399,E2 -16009.399} C_VEL
LIN {X 0,Y 305.817,Z 174.392,A -85,B 0,C 180,E1 -16012.074,E2 -16012.074} C_VEL
LIN {X 0,Y 305.694,Z 174.409,A -85,B 0,C 180,E1 -16014.723,E2 -16014.723} C_VEL
LIN {X 0,Y 305.961,Z 174.375,A -85,B 0,C 180,E1 -16018.683,E2 -16018.683} C_VEL
LIN {X 0,Y 305.961,Z 174.373,A -85,B 0,C 180,E1 -16021.316,E2 -16021.316} C_VEL
LIN {X 0,Y 305.648,Z 174.414,A -85,B 0,C 180,E1 -16023.955,E2 -16023.955} C_VEL
LIN {X 0,Y 306.013,Z 175.771,A -85,B 0,C 180,E1 -16026.627,E2 -16026.627} C_VEL
LIN {X 0,Y 306.015,Z 177.302,A -85,B 0,C 180,E1 -16029.25,E2 -16029.25} C_VEL
LIN {X 0,Y 305.733,Z 179.895,A -85,B 0,C 180,E1 -16033.289,E2 -16033.289} C_VEL
LIN {X 0,Y 305.358,Z 182.749,A -85,B 0,C 180,E1 -16037.409,E2 -16037.409} C_VEL
LIN {X 0,Y 305.158,Z 184.615,A -85,B 0,C 180,E1 -16039.974,E2 -16039.974} C_VEL
LIN {X 0,Y 306.306,Z 187.844,A -85,B 0,C 180,E1 -16040.261,E2 -16040.261} C_VEL
LIN {X 0,Y 310.633,Z 199.401,A -85,B 0,C 180,E1 -16041.396,E2 -16041.396} C_VEL
LIN {X 0,Y 313.731,Z 210.173,A -85,B 0,C 180,E1 -16042.558,E2 -16042.558} C_VEL
LIN {X 0,Y 315.409,Z 217.964,A -85,B 0,C 180,E1 -16043.471,E2 -16043.471} C_VEL
LIN {X 0,Y 315.09,Z 222.901,A -85,B 0,C 180,E1 -16043.984,E2 -16043.984} C_VEL
LIN {X 0,Y 313.422,Z 234.516,A -85,B 0,C 180,E1 -16045.345,E2 -16045.345} C_VEL
LIN {X 0,Y 311.756,Z 245.344,A -85,B 0,C 180,E1 -16046.979,E2 -16046.979} C_VEL
LIN {X 0,Y 310.024,Z 255.002,A -85,B 0,C 180,E1 -16048.797,E2 -16048.797} C_VEL
LIN {X 0,Y 308.723,Z 262.087,A -85,B 0,C 180,E1 -16050.453,E2 -16050.453} C_VEL
LIN {X 0,Y 307.429,Z 268.378,A -85,B 0,C 180,E1 -16052.237,E2 -16052.237} C_VEL
LIN {X 0,Y 306.251,Z 274.136,A -85,B 0,C 180,E1 -16054.295,E2 -16054.295} C_VEL
LIN {X 0,Y 305.257,Z 279.321,A -85,B 0,C 180,E1 -16056.769,E2 -16056.769} C_VEL
LIN {X 0,Y 304.653,Z 281.996,A -85,B 0,C 180,E1 -16058.524,E2 -16058.524} C_VEL
LIN {X 0,Y 304.215,Z 283.955,A -85,B 0,C 180,E1 -16060.326,E2 -16060.326} C_VEL
LIN {X 0,Y 303.912,Z 285.205,A -85,B 0,C 180,E1 -16062.268,E2 -16062.268} C_VEL
LIN {X 0,Y 303.735,Z 285.57,A -85,B 0,C 180,E1 -16064.168,E2 -16064.168} C_VEL
LIN {X 0,Y 303.689,Z 285.124,A -85,B 0,C 180,E1 -16066.031,E2 -16066.031} C_VEL
LIN {X 0,Y 303.818,Z 283.915,A -85,B 0,C 180,E1 -16067.868,E2 -16067.868} C_VEL
LIN {X 0,Y 304.119,Z 281.936,A -85,B 0,C 180,E1 -16069.694,E2 -16069.694} C_VEL
LIN {X 0,Y 304.538,Z 278.818,A -85,B 0,C 180,E1 -16071.686,E2 -16071.686} C_VEL
LIN {X 0,Y 305.064,Z 274.481,A -85,B 0,C 180,E1 -16073.737,E2 -16073.737} C_VEL
LIN {X 0,Y 305.798,Z 268.737,A -85,B 0,C 180,E1 -16075.828,E2 -16075.828} C_VEL
LIN {X 0,Y 306.801,Z 261.351,A -85,B 0,C 180,E1 -16077.947,E2 -16077.947} C_VEL
LIN {X 0,Y 308.029,Z 252.9,A -85,B 0,C 180,E1 -16079.87,E2 -16079.87} C_VEL
LIN {X 0,Y 309.308,Z 242.873,A -85,B 0,C 180,E1 -16081.7,E2 -16081.7} C_VEL
LIN {X 0,Y 310.575,Z 232.229,A -85,B 0,C 180,E1 -16083.258,E2 -16083.258} C_VEL
LIN {X 0,Y 311.766,Z 221.286,A -85,B 0,C 180,E1 -16084.53,E2 -16084.53} C_VEL
LIN {X 0,Y 312.472,Z 213.994,A -85,B 0,C 180,E1 -16085.234,E2 -16085.234} C_VEL
LIN {X 0,Y 310.271,Z 203.077,A -85,B 0,C 180,E1 -16086.293,E2 -16086.293} C_VEL
LIN {X 0,Y 307.072,Z 190.397,A -85,B 0,C 180,E1 -16087.301,E2 -16087.301} C_VEL
LIN {X 0,Y 304.513,Z 181.296,A -85,B 0,C 180,E1 -16087.911,E2 -16087.911} C_VEL
LIN {X 0,Y 304.648,Z 178.411,A -85,B 0,C 180,E1 -16091.157,E2 -16091.157} C_VEL
LIN {X 0,Y 304.904,Z 174.666,A -85,B 0,C 180,E1 -16095.484,E2 -16095.484} C_VEL
LIN {X 0,Y 305.385,Z 174.442,A -85,B 0,C 180,E1 -16099.391,E2 -16099.391} C_VEL
LIN {X 0,Y 305.761,Z 174.4,A -85,B 0,C 180,E1 -16102.073,E2 -16102.073} C_VEL
LIN {X 0,Y 305.68,Z 174.407,A -85,B 0,C 180,E1 -16104.723,E2 -16104.723} C_VEL
LIN {X 0,Y 305.954,Z 174.372,A -85,B 0,C 180,E1 -16108.684,E2 -16108.684} C_VEL
LIN {X 0,Y 305.954,Z 174.371,A -85,B 0,C 180,E1 -16111.316,E2 -16111.316} C_VEL
LIN {X 0,Y 305.849,Z 174.385,A -85,B 0,C 180,E1 -16116.597,E2 -16116.597} C_VEL
LIN {X 0,Y 305.732,Z 174.4,A -85,B 0,C 180,E1 -16119.26,E2 -16119.26} C_VEL
LIN {X 0,Y 305.585,Z 174.419,A -85,B 0,C 180,E1 -16123.296,E2 -16123.296} C_VEL
LIN {X 0,Y 305.59,Z 174.419,A -85,B 0,C 180,E1 -16126.02,E2 -16126.02} C_VEL
LIN {X 0,Y 305.573,Z 174.422,A -85,B 0,C 180,E1 -16129.445,E2 -16129.445} C_VEL
LIN {X 0,Y 305.487,Z 174.431,A -85,B 0,C 180,E1 -16133.042,E2 -16133.042} C_VEL
LIN {X 0,Y 305.522,Z 174.424,A -85,B 0,C 180,E1 -16136.219,E2 -16136.219} C_VEL
LIN {X 0,Y 305.485,Z 174.432,A -85,B 0,C 180,E1 -16139.048,E2 -16139.048} C_VEL
LIN {X 0,Y 305.438,Z 174.436,A -85,B 0,C 180,E1 -16141.953,E2 -16141.953} C_VEL
LIN {X 0,Y 305.459,Z 174.436,A -85,B 0,C 180,E1 -16145.113,E2 -16145.113} C_VEL
LIN {X 0,Y 305.437,Z 174.435,A -85,B 0,C 180,E1 -16148.527,E2 -16148.527} C_VEL
LIN {X 0,Y 305.456,Z 174.435,A -85,B 0,C 180,E1 -16152.587,E2 -16152.587} C_VEL
LIN {X 0,Y 305.44,Z 174.435,A -85,B 0,C 180,E1 -16156.349,E2 -16156.349} C_VEL
LIN {X 0,Y 305.455,Z 174.432,A -85,B 0,C 180,E1 -16159.893,E2 -16159.893} C_VEL
LIN {X 0,Y 305.478,Z 174.431,A -85,B 0,C 180,E1 -16163.632,E2 -16163.632} C_VEL
LIN {X 0,Y 305.463,Z 174.435,A -85,B 0,C 180,E1 -16166.484,E2 -16166.484} C_VEL
LIN {X 0,Y 305.456,Z 174.432,A -85,B 0,C 180,E1 -16169.591,E2 -16169.591} C_VEL
LIN {X 0,Y 305.513,Z 174.429,A -85,B 0,C 180,E1 -16172.609,E2 -16172.609} C_VEL
LIN {X 0,Y 305.507,Z 174.426,A -85,B 0,C 180,E1 -16175.539,E2 -16175.539} C_VEL
LIN {X 0,Y 305.519,Z 174.426,A -85,B 0,C 180,E1 -16179.816,E2 -16179.816} C_VEL
LIN {X 0,Y 305.574,Z 174.42,A -85,B 0,C 180,E1 -16182.604,E2 -16182.604} C_VEL
LIN {X 0,Y 305.649,Z 174.407,A -85,B 0,C 180,E1 -16185.35,E2 -16185.35} C_VEL
LIN {X 0,Y 305.596,Z 174.417,A -85,B 0,C 180,E1 -16187.943,E2 -16187.943} C_VEL
LIN {X 0,Y 305.014,Z 174.495,A -85,B 0,C 180,E1 -16189.045,E2 -16189.045} C_VEL
LIN {X 0,Y 302.291,Z 174.834,A -85,B 0,C 180,E1 -16190.842,E2 -16190.842} C_VEL
LIN {X 0,Y 299.082,Z 175.228,A -85,B 0,C 180,E1 -16193.045,E2 -16193.045} C_VEL
LIN {X 0,Y 298.713,Z 175.271,A -85,B 0,C 180,E1 -16193.806,E2 -16193.806} C_VEL
LIN {X 0,Y 298.924,Z 175.246,A -85,B 0,C 180,E1 -16198.653,E2 -16198.653} C_VEL
LIN {X 0,Y 298.923,Z 175.247,A -85,B 0,C 180,E1 -16201.348,E2 -16201.348} C_VEL
LIN {X 0,Y 298.644,Z 175.283,A -85,B 0,C 180,E1 -16205.402,E2 -16205.402} C_VEL
LIN {X 0,Y 298.714,Z 175.274,A -85,B 0,C 180,E1 -16208.116,E2 -16208.116} C_VEL
LIN {X 0,Y 298.552,Z 175.295,A -85,B 0,C 180,E1 -16212.232,E2 -16212.232} C_VEL
LIN {X 0,Y 298.607,Z 175.288,A -85,B 0,C 180,E1 -16215.21,E2 -16215.21} C_VEL
LIN {X 0,Y 298.542,Z 175.295,A -85,B 0,C 180,E1 -16219.244,E2 -16219.244} C_VEL
LIN {X 0,Y 298.459,Z 175.31,A -85,B 0,C 180,E1 -16223.598,E2 -16223.598} C_VEL
LIN {X 0,Y 298.487,Z 175.302,A -85,B 0,C 180,E1 -16226.575,E2 -16226.575} C_VEL
LIN {X 0,Y 298.418,Z 175.313,A -85,B 0,C 180,E1 -16229.642,E2 -16229.642} C_VEL
LIN {X 0,Y 298.397,Z 175.314,A -85,B 0,C 180,E1 -16232.801,E2 -16232.801} C_VEL
LIN {X 0,Y 298.448,Z 175.309,A -85,B 0,C 180,E1 -16236.808,E2 -16236.808} C_VEL
LIN {X 0,Y 298.436,Z 175.426,A -85,B 0,C 180,E1 -16240.324,E2 -16240.324} C_VEL
LIN {X 0,Y 299.126,Z 179.089,A -85,B 0,C 180,E1 -16243.252,E2 -16243.252} C_VEL
LIN {X 0,Y 300.078,Z 184.326,A -85,B 0,C 180,E1 -16247.219,E2 -16247.219} C_VEL
LIN {X 0,Y 301.002,Z 189.529,A -85,B 0,C 180,E1 -16250.919,E2 -16250.919} C_VEL
LIN {X 0,Y 301.244,Z 192.098,A -85,B 0,C 180,E1 -16252.658,E2 -16252.658} C_VEL
LIN {X 0,Y 300.76,Z 197.138,A -85,B 0,C 180,E1 -16255.888,E2 -16255.888} C_VEL
LIN {X 0,Y 299.563,Z 204.242,A -85,B 0,C 180,E1 -16260.234,E2 -16260.234} C_VEL
LIN {X 0,Y 298.655,Z 210.864,A -85,B 0,C 180,E1 -16264.193,E2 -16264.193} C_VEL
LIN {X 0,Y 298.259,Z 214.309,A -85,B 0,C 180,E1 -16266.22,E2 -16266.22} C_VEL
LIN {X 0,Y 300.667,Z 228.221,A -85,B 0,C 180,E1 -16267.021,E2 -16267.021} C_VEL
LIN {X 0,Y 302.456,Z 241.293,A -85,B 0,C 180,E1 -16268.03,E2 -16268.03} C_VEL
LIN {X 0,Y 303.63,Z 253.905,A -85,B 0,C 180,E1 -16269.25,E2 -16269.25} C_VEL
LIN {X 0,Y 304.063,Z 260.977,A -85,B 0,C 180,E1 -16270.067,E2 -16270.067} C_VEL
LIN {X 0,Y 302.39,Z 272.451,A -85,B 0,C 180,E1 -16271.539,E2 -16271.539} C_VEL
LIN {X 0,Y 301.126,Z 282.23,A -85,B 0,C 180,E1 -16273.12,E2 -16273.12} C_VEL
LIN {X 0,Y 299.692,Z 291.803,A -85,B 0,C 180,E1 -16275.051,E2 -16275.051} C_VEL
LIN {X 0,Y 298.52,Z 299.858,A -85,B 0,C 180,E1 -16277.076,E2 -16277.076} C_VEL
LIN {X 0,Y 297.696,Z 306.325,A -85,B 0,C 180,E1 -16279.114,E2 -16279.114} C_VEL
LIN {X 0,Y 297.104,Z 311.444,A -85,B 0,C 180,E1 -16281.155,E2 -16281.155} C_VEL
LIN {X 0,Y 296.794,Z 315.406,A -85,B 0,C 180,E1 -16283.201,E2 -16283.201} C_VEL
LIN {X 0,Y 296.701,Z 317.434,A -85,B 0,C 180,E1 -16284.563,E2 -16284.563} C_VEL
LIN {X 0,Y 296.688,Z 319.039,A -85,B 0,C 180,E1 -16285.925,E2 -16285.925} C_VEL
LIN {X 0,Y 296.632,Z 320.224,A -85,B 0,C 180,E1 -16287.284,E2 -16287.284} C_VEL
LIN {X 0,Y 296.669,Z 320.962,A -85,B 0,C 180,E1 -16288.643,E2 -16288.643} C_VEL
LIN {X 0,Y 296.777,Z 321.292,A -85,B 0,C 180,E1 -16290,E2 -16290} C_VEL
LIN {X 0,Y 296.62,Z 320.743,A -85,B 0,C 180,E1 -16292.716,E2 -16292.716} C_VEL
LIN {X 0,Y 296.639,Z 319.84,A -85,B 0,C 180,E1 -16294.076,E2 -16294.076} C_VEL
LIN {X 0,Y 296.703,Z 318.099,A -85,B 0,C 180,E1 -16295.81,E2 -16295.81} C_VEL
LIN {X 0,Y 296.965,Z 314.648,A -85,B 0,C 180,E1 -16298.164,E2 -16298.164} C_VEL
LIN {X 0,Y 297.459,Z 310.527,A -85,B 0,C 180,E1 -16300.207,E2 -16300.207} C_VEL
LIN {X 0,Y 298.419,Z 304.254,A -85,B 0,C 180,E1 -16302.583,E2 -16302.583} C_VEL
LIN {X 0,Y 299.67,Z 297.47,A -85,B 0,C 180,E1 -16304.603,E2 -16304.603} C_VEL
LIN {X 0,Y 301.147,Z 289.318,A -85,B 0,C 180,E1 -16306.565,E2 -16306.565} C_VEL
LIN {X 0,Y 302.579,Z 280.658,A -85,B 0,C 180,E1 -16308.274,E2 -16308.274} C_VEL
LIN {X 0,Y 304.455,Z 270.318,A -85,B 0,C 180,E1 -16309.907,E2 -16309.907} C_VEL
LIN {X 0,Y 305.629,Z 262.982,A -85,B 0,C 180,E1 -16310.881,E2 -16310.881} C_VEL
LIN {X 0,Y 305.393,Z 250.6,A -85,B 0,C 180,E1 -16312.383,E2 -16312.383} C_VEL
LIN {X 0,Y 304.533,Z 239.206,A -85,B 0,C 180,E1 -16313.547,E2 -16313.547} C_VEL
LIN {X 0,Y 302.257,Z 226.073,A -85,B 0,C 180,E1 -16314.742,E2 -16314.742} C_VEL
LIN {X 0,Y 298.805,Z 212.523,A -85,B 0,C 180,E1 -16315.807,E2 -16315.807} C_VEL
LIN {X 0,Y 298.747,Z 211.917,A -85,B 0,C 180,E1 -16315.843,E2 -16315.843} C_VEL
LIN {X 0,Y 299.684,Z 205.52,A -85,B 0,C 180,E1 -16319.806,E2 -16319.806} C_VEL
LIN {X 0,Y 300.704,Z 200.104,A -85,B 0,C 180,E1 -16323.314,E2 -16323.314} C_VEL
LIN {X 0,Y 301.485,Z 195.502,A -85,B 0,C 180,E1 -16326.473,E2 -16326.473} C_VEL
LIN {X 0,Y 301.574,Z 193.969,A -85,B 0,C 180,E1 -16327.593,E2 -16327.593} C_VEL
LIN {X 0,Y 301.034,Z 189.909,A -85,B 0,C 180,E1 -16330.821,E2 -16330.821} C_VEL
LIN {X 0,Y 300.266,Z 185.672,A -85,B 0,C 180,E1 -16334.602,E2 -16334.602} C_VEL
LIN {X 0,Y 299.822,Z 183.052,A -85,B 0,C 180,E1 -16337.173,E2 -16337.173} C_VEL
LIN {X 0,Y 299.228,Z 179.805,A -85,B 0,C 180,E1 -16340.812,E2 -16340.812} C_VEL
LIN {X 0,Y 298.795,Z 177.341,A -85,B 0,C 180,E1 -16343.982,E2 -16343.982} C_VEL
LIN {X 0,Y 298.399,Z 175.313,A -85,B 0,C 180,E1 -16347.2,E2 -16347.2} C_VEL
LIN {X 0,Y 298.431,Z 175.311,A -85,B 0,C 180,E1 -16350.616,E2 -16350.616} C_VEL
LIN {X 0,Y 298.482,Z 175.302,A -85,B 0,C 180,E1 -16353.476,E2 -16353.476} C_VEL
LIN {X 0,Y 298.44,Z 175.311,A -85,B 0,C 180,E1 -16356.697,E2 -16356.697} C_VEL
LIN {X 0,Y 298.524,Z 175.302,A -85,B 0,C 180,E1 -16360.755,E2 -16360.755} C_VEL
LIN {X 0,Y 298.589,Z 175.292,A -85,B 0,C 180,E1 -16364.994,E2 -16364.994} C_VEL
LIN {X 0,Y 298.598,Z 175.293,A -85,B 0,C 180,E1 -16369.146,E2 -16369.146} C_VEL
LIN {X 0,Y 298.763,Z 175.271,A -85,B 0,C 180,E1 -16371.885,E2 -16371.885} C_VEL
LIN {X 0,Y 298.665,Z 175.284,A -85,B 0,C 180,E1 -16374.598,E2 -16374.598} C_VEL
LIN {X 0,Y 298.928,Z 175.251,A -85,B 0,C 180,E1 -16378.652,E2 -16378.652} C_VEL
LIN {X 0,Y 298.927,Z 175.25,A -85,B 0,C 180,E1 -16381.346,E2 -16381.346} C_VEL
LIN {X 0,Y 298.84,Z 175.261,A -85,B 0,C 180,E1 -16382.695,E2 -16382.695} C_VEL
LIN {X 0,Y 299.036,Z 177.156,A -85,B 0,C 180,E1 -16386.748,E2 -16386.748} C_VEL
LIN {X 0,Y 298.993,Z 178.71,A -85,B 0,C 180,E1 -16389.47,E2 -16389.47} C_VEL
LIN {X 0,Y 298.691,Z 181.311,A -85,B 0,C 180,E1 -16393.608,E2 -16393.608} C_VEL
LIN {X 0,Y 298.423,Z 183.195,A -85,B 0,C 180,E1 -16396.415,E2 -16396.415} C_VEL
LIN {X 0,Y 298.209,Z 185.128,A -85,B 0,C 180,E1 -16399.175,E2 -16399.175} C_VEL
LIN {X 0,Y 300.573,Z 191.284,A -85,B 0,C 180,E1 -16399.789,E2 -16399.789} C_VEL
LIN {X 0,Y 304.914,Z 203.293,A -85,B 0,C 180,E1 -16401.078,E2 -16401.078} C_VEL
LIN {X 0,Y 307.746,Z 213.966,A -85,B 0,C 180,E1 -16402.312,E2 -16402.312} C_VEL
LIN {X 0,Y 308.98,Z 220.298,A -85,B 0,C 180,E1 -16403.101,E2 -16403.101} C_VEL
LIN {X 0,Y 307.629,Z 230.796,A -85,B 0,C 180,E1 -16404.281,E2 -16404.281} C_VEL
LIN {X 0,Y 306.002,Z 240.936,A -85,B 0,C 180,E1 -16405.689,E2 -16405.689} C_VEL
LIN {X 0,Y 304.495,Z 249.556,A -85,B 0,C 180,E1 -16407.157,E2 -16407.157} C_VEL
LIN {X 0,Y 302.835,Z 258.113,A -85,B 0,C 180,E1 -16408.938,E2 -16408.938} C_VEL
LIN {X 0,Y 301.305,Z 265.621,A -85,B 0,C 180,E1 -16410.873,E2 -16410.873} C_VEL
LIN {X 0,Y 299.859,Z 272.189,A -85,B 0,C 180,E1 -16413.019,E2 -16413.019} C_VEL
LIN {X 0,Y 298.767,Z 277.525,A -85,B 0,C 180,E1 -16415.297,E2 -16415.297} C_VEL
LIN {X 0,Y 298.203,Z 280.209,A -85,B 0,C 180,E1 -16416.744,E2 -16416.744} C_VEL
LIN {X 0,Y 297.523,Z 283.061,A -85,B 0,C 180,E1 -16418.783,E2 -16418.783} C_VEL
LIN {X 0,Y 296.905,Z 285.339,A -85,B 0,C 180,E1 -16421.511,E2 -16421.511} C_VEL
LIN {X 0,Y 296.694,Z 285.971,A -85,B 0,C 180,E1 -16423.388,E2 -16423.388} C_VEL
LIN {X 0,Y 296.608,Z 285.828,A -85,B 0,C 180,E1 -16425.302,E2 -16425.302} C_VEL
LIN {X 0,Y 296.658,Z 284.827,A -85,B 0,C 180,E1 -16427.256,E2 -16427.256} C_VEL
LIN {X 0,Y 296.934,Z 282.951,A -85,B 0,C 180,E1 -16429.234,E2 -16429.234} C_VEL
LIN {X 0,Y 297.344,Z 280.092,A -85,B 0,C 180,E1 -16431.258,E2 -16431.258} C_VEL
LIN {X 0,Y 297.858,Z 276.078,A -85,B 0,C 180,E1 -16433.343,E2 -16433.343} C_VEL
LIN {X 0,Y 298.619,Z 270.352,A -85,B 0,C 180,E1 -16435.608,E2 -16435.608} C_VEL
LIN {X 0,Y 299.55,Z 263.785,A -85,B 0,C 180,E1 -16437.63,E2 -16437.63} C_VEL
LIN {X 0,Y 300.864,Z 254.896,A -85,B 0,C 180,E1 -16439.801,E2 -16439.801} C_VEL
LIN {X 0,Y 302.121,Z 245.797,A -85,B 0,C 180,E1 -16441.583,E2 -16441.583} C_VEL
LIN {X 0,Y 303.34,Z 235.95,A -85,B 0,C 180,E1 -16443.141,E2 -16443.141} C_VEL
LIN {X 0,Y 304.726,Z 224.273,A -85,B 0,C 180,E1 -16444.622,E2 -16444.622} C_VEL
LIN {X 0,Y 305.647,Z 215.145,A -85,B 0,C 180,E1 -16445.55,E2 -16445.55} C_VEL
LIN {X 0,Y 303.123,Z 202.686,A -85,B 0,C 180,E1 -16446.787,E2 -16446.787} C_VEL
LIN {X 0,Y 299.62,Z 189.389,A -85,B 0,C 180,E1 -16447.857,E2 -16447.857} C_VEL
